Yaskawa INFORM job: DEMO_ROOF_SIDE_0625_3PAINT_54.JBI

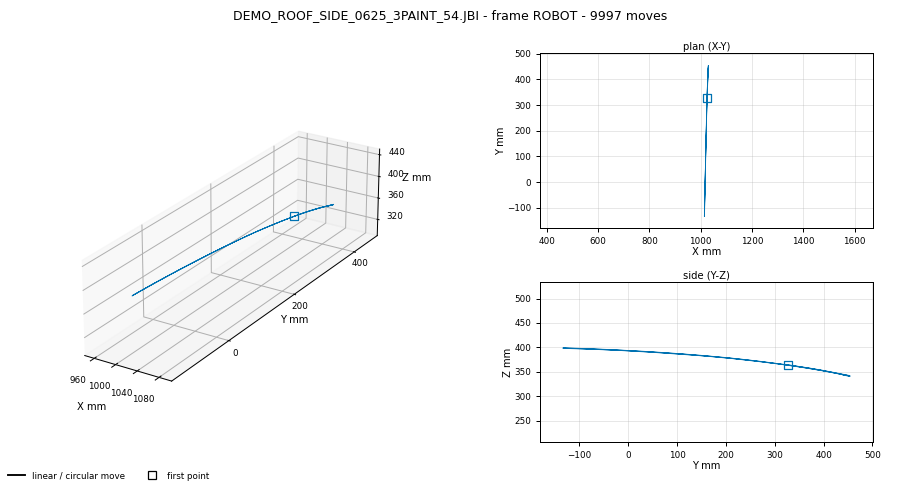
[picture p0: tool path of DEMO_ROOF_SIDE_0625_3PAINT_54.JBI in frame ROBOT, 9997 of 9997 moves have a stored position in this frame; points joined in program order, loops and branches not executed]
/JOB
//NAME DEMO_ROOF_SIDE_0625_3PAINT54
//POS
///NPOS 9997,0,0,0,0,0
///TOOL 0
///USER 0
///POSTYPE ROBOT
///RECTAN
///RCONF 1,0,0,0,0,0,0,0,0,0,0,0,0,0,0,0,0,0,0,0,0,0,0,0
C00000=1025.330,327.745,364.272,171.208,47.893,159.349
C00001=1025.337,327.993,364.236,171.213,47.892,159.350
C00002=1025.345,328.240,364.202,171.218,47.891,159.350
C00003=1025.352,328.488,364.166,171.225,47.891,159.351
C00004=1025.359,328.735,364.131,171.230,47.890,159.352
C00005=1025.365,328.982,364.095,171.237,47.889,159.352
C00006=1025.373,329.230,364.060,171.242,47.888,159.353
C00007=1025.380,329.477,364.025,171.248,47.888,159.354
C00008=1025.388,329.725,363.990,171.254,47.886,159.354
C00009=1025.395,329.972,363.954,171.260,47.886,159.355
C00010=1025.402,330.219,363.919,171.265,47.885,159.355
C00011=1025.409,330.467,363.883,171.272,47.885,159.356
C00012=1025.417,330.714,363.848,171.277,47.884,159.357
C00013=1025.424,330.961,363.813,171.284,47.883,159.358
C00014=1025.431,331.209,363.778,171.289,47.883,159.358
C00015=1025.438,331.456,363.742,171.295,47.882,159.359
C00016=1025.445,331.704,363.706,171.301,47.881,159.359
C00017=1025.453,331.951,363.672,171.307,47.880,159.360
C00018=1025.461,332.199,363.635,171.313,47.880,159.361
C00019=1025.467,332.446,363.600,171.319,47.880,159.361
C00020=1025.475,332.693,363.564,171.325,47.878,159.362
C00021=1025.482,332.941,363.529,171.331,47.878,159.363
C00022=1025.489,333.188,363.493,171.337,47.877,159.363
C00023=1025.497,333.435,363.458,171.343,47.877,159.364
C00024=1025.505,333.683,363.422,171.348,47.876,159.365
C00025=1025.512,333.929,363.386,171.355,47.876,159.365
C00026=1025.519,334.177,363.351,171.361,47.875,159.366
C00027=1025.526,334.424,363.315,171.368,47.875,159.367
C00028=1025.534,334.672,363.279,171.373,47.874,159.368
C00029=1025.540,334.920,363.242,171.380,47.873,159.368
C00030=1025.547,335.167,363.207,171.385,47.873,159.369
C00031=1025.555,335.414,363.170,171.392,47.873,159.370
C00032=1025.562,335.661,363.135,171.398,47.872,159.371
C00033=1025.574,336.048,363.078,171.407,47.871,159.372
C00034=1025.586,336.435,363.022,171.416,47.871,159.373
C00035=1025.597,336.822,362.966,171.426,47.870,159.374
C00036=1025.608,337.209,362.909,171.435,47.869,159.375
C00037=1025.616,337.456,362.873,171.442,47.869,159.376
C00038=1025.623,337.704,362.837,171.448,47.869,159.376
C00039=1025.631,337.951,362.801,171.455,47.868,159.377
C00040=1025.638,338.198,362.765,171.460,47.868,159.378
C00041=1025.646,338.446,362.728,171.467,47.867,159.379
C00042=1025.654,338.693,362.692,171.474,47.867,159.380
C00043=1025.661,338.940,362.656,171.479,47.866,159.380
C00044=1025.668,339.187,362.620,171.486,47.866,159.381
C00045=1025.676,339.435,362.584,171.492,47.866,159.382
C00046=1025.684,339.682,362.548,171.498,47.865,159.383
C00047=1025.691,339.930,362.511,171.504,47.865,159.383
C00048=1025.698,340.176,362.474,171.511,47.865,159.384
C00049=1025.706,340.423,362.438,171.517,47.865,159.385
C00050=1025.713,340.671,362.402,171.523,47.864,159.386
C00051=1025.721,340.918,362.364,171.530,47.864,159.387
C00052=1025.728,341.165,362.328,171.536,47.864,159.387
C00053=1025.735,341.412,362.292,171.543,47.864,159.388
C00054=1025.743,341.659,362.255,171.548,47.863,159.389
C00055=1025.750,341.907,362.218,171.555,47.863,159.390
C00056=1025.758,342.154,362.182,171.561,47.863,159.391
C00057=1025.765,342.401,362.145,171.568,47.863,159.392
C00058=1025.773,342.649,362.109,171.575,47.862,159.392
C00059=1025.781,342.896,362.072,171.581,47.863,159.393
C00060=1025.788,343.143,362.035,171.587,47.862,159.394
C00061=1025.796,343.390,361.998,171.593,47.862,159.395
C00062=1025.803,343.638,361.962,171.600,47.862,159.396
C00063=1025.811,343.885,361.924,171.607,47.861,159.397
C00064=1025.818,344.131,361.888,171.613,47.862,159.397
C00065=1025.825,344.379,361.851,171.619,47.861,159.398
C00066=1025.833,344.625,361.814,171.626,47.861,159.399
C00067=1025.841,344.872,361.777,171.632,47.861,159.400
C00068=1025.848,345.120,361.740,171.639,47.861,159.401
C00069=1025.856,345.367,361.703,171.645,47.861,159.402
C00070=1025.864,345.615,361.665,171.652,47.861,159.403
C00071=1025.871,345.862,361.629,171.658,47.860,159.403
C00072=1025.879,346.109,361.591,171.664,47.861,159.404
C00073=1025.887,346.356,361.555,171.671,47.861,159.405
C00074=1025.895,346.603,361.518,171.678,47.860,159.406
C00075=1025.902,346.850,361.480,171.685,47.860,159.407
C00076=1025.910,347.097,361.443,171.691,47.861,159.408
C00077=1025.917,347.345,361.406,171.698,47.860,159.409
C00078=1025.925,347.591,361.369,171.705,47.860,159.410
C00079=1025.932,347.839,361.332,171.711,47.861,159.411
C00080=1025.941,348.086,361.295,171.718,47.861,159.412
C00081=1025.948,348.333,361.257,171.725,47.860,159.412
C00082=1025.956,348.580,361.220,171.732,47.860,159.413
C00083=1025.963,348.827,361.182,171.738,47.861,159.414
C00084=1025.971,349.074,361.144,171.745,47.861,159.415
C00085=1025.979,349.321,361.107,171.752,47.861,159.416
C00086=1025.986,349.568,361.070,171.758,47.861,159.417
C00087=1025.994,349.816,361.032,171.765,47.861,159.418
C00088=1026.005,350.185,360.975,171.775,47.861,159.420
C00089=1026.016,350.531,360.923,171.784,47.861,159.421
C00090=1026.023,350.754,360.890,171.790,47.862,159.422
C00091=1026.030,350.977,360.855,171.796,47.862,159.423
C00092=1026.037,351.199,360.821,171.802,47.862,159.424
C00093=1026.044,351.423,360.787,171.809,47.862,159.424
C00094=1026.051,351.645,360.753,171.815,47.862,159.425
C00095=1026.058,351.868,360.719,171.821,47.863,159.426
C00096=1026.065,352.090,360.685,171.827,47.863,159.427
C00097=1026.074,352.338,360.648,171.834,47.863,159.428
C00098=1026.081,352.584,360.609,171.841,47.863,159.429
C00099=1026.088,352.831,360.572,171.848,47.863,159.430
C00100=1026.096,353.079,360.533,171.855,47.863,159.431
C00101=1026.104,353.325,360.496,171.861,47.864,159.432
C00102=1026.113,353.573,360.458,171.869,47.864,159.433
C00103=1026.120,353.820,360.420,171.876,47.864,159.434
C00104=1026.128,354.066,360.382,171.883,47.864,159.435
C00105=1026.136,354.314,360.345,171.890,47.865,159.436
C00106=1026.144,354.560,360.306,171.897,47.865,159.437
C00107=1026.152,354.808,360.268,171.904,47.865,159.438
C00108=1026.160,355.054,360.231,171.910,47.866,159.439
C00109=1026.168,355.302,360.192,171.917,47.866,159.440
C00110=1026.175,355.548,360.154,171.924,47.866,159.441
C00111=1026.184,355.795,360.115,171.932,47.867,159.442
C00112=1026.191,356.042,360.077,171.939,47.867,159.443
C00113=1026.199,356.289,360.038,171.946,47.868,159.445
C00114=1026.206,356.536,360.001,171.953,47.868,159.446
C00115=1026.215,356.783,359.962,171.960,47.868,159.447
C00116=1026.222,357.030,359.924,171.967,47.868,159.448
C00117=1026.230,357.277,359.885,171.975,47.869,159.449
C00118=1026.239,357.524,359.847,171.981,47.870,159.450
C00119=1026.247,357.771,359.809,171.988,47.870,159.451
C00120=1026.255,358.018,359.771,171.995,47.871,159.452
C00121=1026.263,358.265,359.732,172.002,47.871,159.453
C00122=1026.271,358.511,359.693,172.010,47.872,159.454
C00123=1026.279,358.758,359.654,172.017,47.872,159.456
C00124=1026.287,359.005,359.616,172.024,47.873,159.457
C00125=1026.295,359.252,359.578,172.031,47.873,159.458
C00126=1026.303,359.499,359.539,172.039,47.874,159.459
C00127=1026.311,359.746,359.500,172.046,47.874,159.460
C00128=1026.319,359.992,359.461,172.053,47.875,159.461
C00129=1026.327,360.239,359.423,172.060,47.875,159.462
C00130=1026.335,360.487,359.384,172.068,47.876,159.463
C00131=1026.344,360.733,359.345,172.075,47.876,159.465
C00132=1026.351,360.980,359.307,172.083,47.877,159.466
C00133=1026.359,361.227,359.267,172.090,47.878,159.467
C00134=1026.367,361.474,359.228,172.097,47.878,159.468
C00135=1026.376,361.720,359.189,172.105,47.879,159.469
C00136=1026.383,361.967,359.151,172.112,47.880,159.470
C00137=1026.391,362.214,359.111,172.119,47.880,159.472
C00138=1026.399,362.461,359.072,172.127,47.881,159.473
C00139=1026.407,362.708,359.033,172.134,47.882,159.474
C00140=1026.416,362.954,358.993,172.143,47.882,159.475
C00141=1026.423,363.202,358.954,172.150,47.883,159.476
C00142=1026.432,363.448,358.915,172.157,47.884,159.478
C00143=1026.440,363.694,358.876,172.165,47.884,159.479
C00144=1026.448,363.941,358.837,172.172,47.885,159.480
C00145=1026.456,364.188,358.798,172.180,47.886,159.481
C00146=1026.464,364.435,358.758,172.187,47.887,159.483
C00147=1026.472,364.682,358.719,172.194,47.888,159.484
C00148=1026.481,364.928,358.679,172.202,47.888,159.485
C00149=1026.489,365.155,358.644,172.209,47.889,159.486
C00150=1026.495,365.381,358.607,172.216,47.890,159.487
C00151=1026.503,365.606,358.571,172.223,47.891,159.488
C00152=1026.511,365.833,358.535,172.230,47.891,159.490
C00153=1026.518,366.059,358.499,172.237,47.892,159.491
C00154=1026.526,366.284,358.462,172.244,47.893,159.492
C00155=1026.534,366.511,358.427,172.251,47.893,159.493
C00156=1026.542,366.737,358.391,172.259,47.895,159.494
C00157=1026.549,366.984,358.351,172.266,47.895,159.496
C00158=1026.558,367.230,358.311,172.274,47.897,159.497
C00159=1026.567,367.477,358.271,172.281,47.897,159.498
C00160=1026.575,367.723,358.232,172.290,47.898,159.499
C00161=1026.583,367.970,358.192,172.297,47.899,159.501
C00162=1026.592,368.218,358.152,172.305,47.900,159.502
C00163=1026.600,368.464,358.113,172.312,47.901,159.503
C00164=1026.609,368.710,358.073,172.321,47.902,159.505
C00165=1026.617,368.957,358.033,172.328,47.903,159.506
C00166=1026.625,369.204,357.994,172.336,47.903,159.507
C00167=1026.633,369.450,357.953,172.344,47.905,159.509
C00168=1026.642,369.698,357.913,172.352,47.906,159.510
C00169=1026.650,369.943,357.873,172.360,47.907,159.511
C00170=1026.658,370.190,357.833,172.368,47.908,159.513
C00171=1026.667,370.436,357.793,172.375,47.909,159.514
C00172=1026.675,370.684,357.753,172.384,47.910,159.516
C00173=1026.683,370.930,357.712,172.392,47.911,159.517
C00174=1026.692,371.176,357.672,172.399,47.912,159.518
C00175=1026.700,371.423,357.632,172.408,47.913,159.520
C00176=1026.709,371.670,357.592,172.415,47.914,159.521
C00177=1026.717,371.916,357.551,172.423,47.915,159.522
C00178=1026.726,372.163,357.512,172.432,47.917,159.524
C00179=1026.734,372.410,357.471,172.440,47.918,159.525
C00180=1026.742,372.656,357.430,172.447,47.919,159.527
C00181=1026.752,372.903,357.390,172.456,47.920,159.528
C00182=1026.760,373.149,357.349,172.464,47.922,159.529
C00183=1026.768,373.395,357.309,172.472,47.923,159.531
C00184=1026.777,373.643,357.269,172.480,47.924,159.532
C00185=1026.785,373.889,357.228,172.488,47.926,159.534
C00186=1026.794,374.135,357.188,172.497,47.926,159.535
C00187=1026.802,374.382,357.147,172.504,47.928,159.537
C00188=1026.811,374.628,357.107,172.513,47.929,159.538
C00189=1026.820,374.875,357.066,172.521,47.930,159.540
C00190=1026.828,375.122,357.025,172.530,47.931,159.541
C00191=1026.838,375.368,356.984,172.537,47.933,159.542
C00192=1026.846,375.614,356.943,172.546,47.934,159.544
C00193=1026.855,375.861,356.903,172.554,47.935,159.545
C00194=1026.863,376.107,356.862,172.563,47.937,159.547
C00195=1026.872,376.354,356.821,172.571,47.938,159.548
C00196=1026.881,376.601,356.781,172.580,47.939,159.550
C00197=1026.890,376.846,356.739,172.588,47.941,159.551
C00198=1026.899,377.093,356.699,172.597,47.942,159.553
C00199=1026.908,377.340,356.658,172.604,47.943,159.554
C00200=1026.916,377.586,356.617,172.613,47.945,159.556
C00201=1026.925,377.833,356.576,172.622,47.946,159.558
C00202=1026.933,378.079,356.534,172.630,47.948,159.559
C00203=1026.942,378.325,356.493,172.639,47.949,159.561
C00204=1026.950,378.572,356.452,172.647,47.951,159.562
C00205=1026.959,378.818,356.410,172.656,47.952,159.564
C00206=1026.967,379.064,356.369,172.664,47.954,159.565
C00207=1026.976,379.311,356.328,172.673,47.955,159.567
C00208=1026.985,379.557,356.286,172.682,47.957,159.569
C00209=1026.994,379.794,356.247,172.690,47.958,159.570
C00210=1027.002,380.030,356.207,172.698,47.960,159.572
C00211=1027.011,380.266,356.167,172.706,47.961,159.573
C00212=1027.018,380.504,356.127,172.714,47.963,159.575
C00213=1027.028,380.741,356.086,172.723,47.964,159.576
C00214=1027.036,380.978,356.047,172.731,47.966,159.578
C00215=1027.045,381.214,356.007,172.739,47.968,159.579
C00216=1027.053,381.450,355.967,172.748,47.969,159.581
C00217=1027.062,381.696,355.925,172.757,47.970,159.583
C00218=1027.071,381.943,355.884,172.766,47.973,159.584
C00219=1027.080,382.189,355.842,172.775,47.974,159.586
C00220=1027.089,382.436,355.800,172.784,47.976,159.588
C00221=1027.098,382.682,355.759,172.793,47.977,159.589
C00222=1027.107,382.928,355.717,172.801,47.979,159.591
C00223=1027.116,383.175,355.675,172.810,47.981,159.593
C00224=1027.125,383.421,355.633,172.819,47.982,159.594
C00225=1027.134,383.667,355.591,172.828,47.984,159.596
C00226=1027.143,383.913,355.549,172.837,47.986,159.598
C00227=1027.152,384.159,355.508,172.845,47.988,159.599
C00228=1027.161,384.407,355.465,172.854,47.989,159.601
C00229=1027.171,384.652,355.423,172.864,47.991,159.603
C00230=1027.180,384.899,355.381,172.873,47.993,159.604
C00231=1027.188,385.145,355.340,172.882,47.995,159.606
C00232=1027.198,385.391,355.297,172.891,47.996,159.608
C00233=1027.207,385.637,355.255,172.900,47.998,159.610
C00234=1027.216,385.884,355.213,172.909,48.001,159.611
C00235=1027.226,386.130,355.172,172.918,48.002,159.613
C00236=1027.235,386.375,355.129,172.927,48.004,159.615
C00237=1027.244,386.622,355.087,172.936,48.006,159.617
C00238=1027.253,386.869,355.044,172.946,48.008,159.618
C00239=1027.263,387.114,355.002,172.955,48.010,159.620
C00240=1027.272,387.360,354.959,172.964,48.012,159.622
C00241=1027.280,387.607,354.917,172.974,48.014,159.624
C00242=1027.290,387.853,354.874,172.983,48.016,159.626
C00243=1027.299,388.099,354.832,172.992,48.018,159.628
C00244=1027.308,388.345,354.789,173.001,48.019,159.629
C00245=1027.318,388.591,354.746,173.011,48.021,159.631
C00246=1027.327,388.837,354.703,173.020,48.023,159.633
C00247=1027.337,389.084,354.661,173.030,48.025,159.635
C00248=1027.346,389.329,354.618,173.039,48.027,159.637
C00249=1027.355,389.575,354.576,173.049,48.030,159.639
C00250=1027.364,389.822,354.532,173.058,48.032,159.640
C00251=1027.373,390.068,354.490,173.067,48.034,159.642
C00252=1027.383,390.314,354.446,173.077,48.036,159.644
C00253=1027.392,390.559,354.403,173.086,48.038,159.646
C00254=1027.402,390.806,354.360,173.097,48.040,159.648
C00255=1027.410,391.052,354.317,173.106,48.042,159.650
C00256=1027.421,391.298,354.274,173.115,48.045,159.652
C00257=1027.430,391.543,354.232,173.125,48.047,159.654
C00258=1027.439,391.790,354.188,173.135,48.049,159.656
C00259=1027.448,392.035,354.145,173.144,48.051,159.658
C00260=1027.458,392.282,354.102,173.155,48.053,159.660
C00261=1027.468,392.528,354.058,173.164,48.055,159.661
C00262=1027.477,392.774,354.016,173.174,48.058,159.664
C00263=1027.486,393.020,353.972,173.183,48.061,159.666
C00264=1027.496,393.266,353.928,173.193,48.063,159.667
C00265=1027.506,393.512,353.885,173.203,48.065,159.669
C00266=1027.515,393.758,353.841,173.213,48.067,159.671
C00267=1027.525,394.004,353.797,173.222,48.070,159.673
C00268=1027.534,394.250,353.755,173.232,48.072,159.675
C00269=1027.544,394.513,353.707,173.243,48.074,159.678
C00270=1027.555,394.776,353.661,173.254,48.077,159.680
C00271=1027.565,395.040,353.615,173.265,48.079,159.682
C00272=1027.575,395.303,353.567,173.275,48.082,159.684
C00273=1027.585,395.549,353.523,173.285,48.084,159.686
C00274=1027.594,395.795,353.480,173.295,48.087,159.688
C00275=1027.604,396.041,353.435,173.305,48.089,159.690
C00276=1027.614,396.287,353.392,173.315,48.092,159.692
C00277=1027.623,396.533,353.348,173.326,48.094,159.694
C00278=1027.633,396.779,353.304,173.336,48.097,159.697
C00279=1027.643,397.025,353.260,173.346,48.100,159.699
C00280=1027.653,397.270,353.216,173.356,48.102,159.701
C00281=1027.663,397.516,353.172,173.366,48.105,159.703
C00282=1027.673,397.762,353.128,173.377,48.107,159.705
C00283=1027.683,398.007,353.084,173.387,48.109,159.707
C00284=1027.692,398.253,353.039,173.398,48.112,159.709
C00285=1027.702,398.499,352.996,173.407,48.115,159.711
C00286=1027.712,398.745,352.951,173.418,48.117,159.713
C00287=1027.721,398.991,352.907,173.428,48.120,159.716
C00288=1027.732,399.236,352.863,173.439,48.122,159.718
C00289=1027.741,399.482,352.818,173.449,48.125,159.720
C00290=1027.751,399.728,352.773,173.460,48.128,159.722
C00291=1027.761,399.974,352.729,173.471,48.130,159.725
C00292=1027.772,400.219,352.684,173.481,48.134,159.727
C00293=1027.781,400.465,352.640,173.491,48.136,159.729
C00294=1027.791,400.711,352.595,173.501,48.139,159.731
C00295=1027.801,400.957,352.550,173.513,48.142,159.733
C00296=1027.811,401.203,352.505,173.523,48.144,159.736
C00297=1027.820,401.448,352.461,173.533,48.147,159.738
C00298=1027.831,401.693,352.416,173.544,48.150,159.740
C00299=1027.841,401.939,352.371,173.555,48.153,159.742
C00300=1027.851,402.185,352.326,173.566,48.155,159.745
C00301=1027.861,402.431,352.282,173.577,48.159,159.747
C00302=1027.871,402.677,352.236,173.588,48.161,159.749
C00303=1027.881,402.922,352.192,173.599,48.164,159.752
C00304=1027.891,403.168,352.146,173.609,48.167,159.754
C00305=1027.901,403.413,352.101,173.620,48.170,159.756
C00306=1027.911,403.659,352.056,173.631,48.173,159.759
C00307=1027.921,403.905,352.011,173.642,48.176,159.761
C00308=1027.931,404.150,351.965,173.653,48.179,159.763
C00309=1027.941,404.396,351.920,173.664,48.182,159.766
C00310=1027.951,404.641,351.875,173.674,48.185,159.768
C00311=1027.962,404.887,351.829,173.686,48.188,159.771
C00312=1027.972,405.133,351.783,173.697,48.191,159.773
C00313=1027.982,405.378,351.739,173.708,48.194,159.775
C00314=1027.993,405.624,351.693,173.719,48.197,159.778
C00315=1028.003,405.870,351.648,173.730,48.200,159.780
C00316=1028.013,406.115,351.602,173.742,48.203,159.783
C00317=1028.024,406.361,351.556,173.753,48.206,159.785
C00318=1028.034,406.606,351.510,173.764,48.209,159.787
C00319=1028.044,406.852,351.465,173.776,48.212,159.790
C00320=1028.055,407.097,351.419,173.787,48.216,159.793
C00321=1028.065,407.343,351.374,173.798,48.219,159.795
C00322=1028.076,407.589,351.328,173.810,48.222,159.797
C00323=1028.086,407.834,351.282,173.821,48.225,159.800
C00324=1028.097,408.080,351.236,173.833,48.228,159.802
C00325=1028.107,408.325,351.190,173.844,48.232,159.805
C00326=1028.118,408.570,351.144,173.855,48.235,159.807
C00327=1028.128,408.816,351.098,173.867,48.237,159.810
C00328=1028.139,409.061,351.053,173.879,48.241,159.812
C00329=1028.151,409.347,350.999,173.892,48.245,159.815
C00330=1028.164,409.633,350.945,173.906,48.249,159.818
C00331=1028.176,409.918,350.891,173.919,48.253,159.821
C00332=1028.189,410.203,350.838,173.933,48.256,159.824
C00333=1028.199,410.448,350.791,173.945,48.260,159.827
C00334=1028.210,410.693,350.745,173.956,48.263,159.830
C00335=1028.221,410.939,350.699,173.969,48.267,159.832
C00336=1028.231,411.184,350.652,173.980,48.270,159.835
C00337=1028.241,411.430,350.606,173.992,48.273,159.838
C00338=1028.252,411.675,350.559,174.005,48.277,159.840
C00339=1028.263,411.921,350.511,174.016,48.281,159.843
C00340=1028.274,412.166,350.466,174.028,48.284,159.846
C00341=1028.284,412.412,350.418,174.041,48.288,159.848
C00342=1028.295,412.657,350.372,174.052,48.291,159.851
C00343=1028.306,412.902,350.325,174.065,48.294,159.854
C00344=1028.317,413.148,350.278,174.077,48.298,159.856
C00345=1028.327,413.393,350.231,174.089,48.302,159.859
C00346=1028.339,413.638,350.184,174.101,48.305,159.862
C00347=1028.349,413.884,350.137,174.114,48.308,159.865
C00348=1028.360,414.129,350.090,174.125,48.312,159.867
C00349=1028.372,414.374,350.043,174.138,48.316,159.870
C00350=1028.382,414.620,349.996,174.150,48.319,159.873
C00351=1028.393,414.865,349.949,174.163,48.324,159.876
C00352=1028.405,415.110,349.902,174.175,48.327,159.879
C00353=1028.415,415.356,349.854,174.188,48.331,159.882
C00354=1028.426,415.601,349.807,174.200,48.334,159.884
C00355=1028.438,415.846,349.760,174.212,48.338,159.887
C00356=1028.449,416.092,349.712,174.225,48.342,159.890
C00357=1028.460,416.337,349.665,174.238,48.346,159.893
C00358=1028.471,416.582,349.617,174.251,48.349,159.896
C00359=1028.482,416.826,349.570,174.263,48.353,159.899
C00360=1028.493,417.072,349.522,174.276,48.357,159.902
C00361=1028.504,417.318,349.474,174.289,48.361,159.905
C00362=1028.516,417.563,349.426,174.302,48.365,159.908
C00363=1028.526,417.807,349.378,174.314,48.369,159.910
C00364=1028.538,418.053,349.331,174.327,48.373,159.913
C00365=1028.549,418.298,349.283,174.340,48.377,159.916
C00366=1028.560,418.544,349.235,174.353,48.381,159.919
C00367=1028.571,418.788,349.187,174.366,48.384,159.922
C00368=1028.583,419.033,349.139,174.379,48.388,159.925
C00369=1028.594,419.279,349.091,174.392,48.392,159.928
C00370=1028.605,419.524,349.043,174.406,48.396,159.931
C00371=1028.617,419.769,348.994,174.419,48.400,159.934
C00372=1028.629,420.014,348.946,174.432,48.405,159.938
C00373=1028.640,420.259,348.898,174.445,48.409,159.941
C00374=1028.651,420.504,348.850,174.459,48.413,159.944
C00375=1028.663,420.749,348.801,174.472,48.417,159.947
C00376=1028.674,420.994,348.753,174.485,48.420,159.950
C00377=1028.686,421.239,348.705,174.498,48.425,159.953
C00378=1028.697,421.484,348.656,174.512,48.429,159.956
C00379=1028.709,421.729,348.607,174.526,48.433,159.959
C00380=1028.721,421.974,348.559,174.539,48.437,159.962
C00381=1028.733,422.219,348.510,174.553,48.442,159.966
C00382=1028.744,422.465,348.462,174.566,48.446,159.969
C00383=1028.755,422.709,348.413,174.580,48.450,159.972
C00384=1028.768,422.954,348.364,174.594,48.454,159.975
C00385=1028.779,423.199,348.315,174.607,48.459,159.978
C00386=1028.791,423.444,348.266,174.622,48.462,159.982
C00387=1028.802,423.689,348.217,174.635,48.467,159.985
C00388=1028.814,423.934,348.168,174.649,48.471,159.988
C00389=1028.828,424.230,348.109,174.666,48.476,159.992
C00390=1028.842,424.525,348.050,174.683,48.482,159.996
C00391=1028.857,424.821,347.990,174.699,48.488,160.000
C00392=1028.871,425.117,347.931,174.717,48.493,160.004
C00393=1028.883,425.361,347.881,174.730,48.497,160.007
C00394=1028.895,425.606,347.832,174.745,48.501,160.011
C00395=1028.907,425.851,347.783,174.759,48.505,160.014
C00396=1028.919,426.096,347.733,174.773,48.510,160.018
C00397=1028.932,426.341,347.684,174.788,48.515,160.021
C00398=1028.943,426.585,347.634,174.802,48.520,160.024
C00399=1028.956,426.830,347.584,174.817,48.524,160.028
C00400=1028.967,427.076,347.534,174.831,48.528,160.031
C00401=1028.979,427.320,347.484,174.846,48.533,160.035
C00402=1028.991,427.565,347.434,174.860,48.538,160.038
C00403=1029.003,427.810,347.384,174.875,48.543,160.042
C00404=1029.015,428.054,347.334,174.890,48.547,160.045
C00405=1029.027,428.298,347.284,174.905,48.552,160.049
C00406=1029.040,428.543,347.234,174.919,48.556,160.052
C00407=1029.052,428.788,347.184,174.933,48.561,160.056
C00408=1029.064,429.033,347.134,174.948,48.566,160.059
C00409=1029.076,429.278,347.084,174.963,48.571,160.063
C00410=1029.089,429.522,347.033,174.978,48.575,160.066
C00411=1029.101,429.766,346.983,174.993,48.580,160.070
C00412=1029.113,430.011,346.933,175.008,48.585,160.074
C00413=1029.125,430.255,346.882,175.023,48.590,160.077
C00414=1029.137,430.500,346.832,175.038,48.595,160.081
C00415=1029.151,430.745,346.781,175.053,48.599,160.085
C00416=1029.163,430.990,346.730,175.070,48.604,160.088
C00417=1029.175,431.234,346.680,175.085,48.609,160.092
C00418=1029.188,431.479,346.630,175.100,48.614,160.096
C00419=1029.200,431.723,346.579,175.115,48.619,160.099
C00420=1029.213,431.967,346.528,175.130,48.624,160.103
C00421=1029.226,432.212,346.477,175.146,48.629,160.107
C00422=1029.239,432.457,346.426,175.162,48.634,160.111
C00423=1029.251,432.701,346.376,175.177,48.639,160.114
C00424=1029.264,432.946,346.325,175.193,48.644,160.118
C00425=1029.277,433.190,346.274,175.209,48.649,160.122
C00426=1029.289,433.435,346.222,175.225,48.654,160.126
C00427=1029.302,433.679,346.171,175.240,48.659,160.130
C00428=1029.315,433.923,346.120,175.257,48.664,160.134
C00429=1029.328,434.168,346.069,175.272,48.669,160.137
C00430=1029.340,434.412,346.016,175.289,48.674,160.141
C00431=1029.354,434.657,345.965,175.304,48.679,160.145
C00432=1029.367,434.901,345.914,175.321,48.685,160.149
C00433=1029.380,435.146,345.863,175.336,48.690,160.153
C00434=1029.392,435.389,345.810,175.352,48.695,160.157
C00435=1029.405,435.634,345.759,175.369,48.700,160.161
C00436=1029.419,435.879,345.707,175.385,48.706,160.165
C00437=1029.431,436.123,345.655,175.401,48.711,160.169
C00438=1029.444,436.367,345.603,175.418,48.716,160.173
C00439=1029.458,436.611,345.551,175.435,48.721,160.177
C00440=1029.471,436.856,345.499,175.451,48.727,160.181
C00441=1029.484,437.099,345.447,175.468,48.732,160.185
C00442=1029.497,437.344,345.395,175.484,48.738,160.190
C00443=1029.510,437.588,345.343,175.501,48.743,160.194
C00444=1029.524,437.832,345.291,175.517,48.748,160.198
C00445=1029.536,438.077,345.239,175.534,48.754,160.202
C00446=1029.550,438.321,345.186,175.552,48.759,160.206
C00447=1029.564,438.565,345.134,175.569,48.765,160.210
C00448=1029.576,438.810,345.082,175.586,48.770,160.215
C00449=1029.590,439.053,345.029,175.603,48.776,160.219
C00450=1029.604,439.296,344.977,175.620,48.781,160.223
C00451=1029.617,439.539,344.925,175.637,48.787,160.227
C00452=1029.630,439.783,344.871,175.654,48.792,160.231
C00453=1029.643,440.026,344.819,175.672,48.798,160.236
C00454=1029.657,440.270,344.767,175.689,48.803,160.240
C00455=1029.671,440.512,344.714,175.706,48.809,160.244
C00456=1029.684,440.756,344.661,175.724,48.815,160.249
C00457=1029.697,441.000,344.608,175.741,48.821,160.253
C00458=1029.712,441.244,344.555,175.759,48.826,160.257
C00459=1029.725,441.488,344.502,175.777,48.832,160.262
C00460=1029.739,441.732,344.449,175.795,48.837,160.266
C00461=1029.753,441.976,344.395,175.812,48.844,160.271
C00462=1029.767,442.219,344.342,175.831,48.849,160.275
C00463=1029.780,442.464,344.289,175.848,48.856,160.280
C00464=1029.794,442.707,344.235,175.866,48.861,160.284
C00465=1029.809,442.950,344.182,175.884,48.867,160.289
C00466=1029.823,443.193,344.129,175.903,48.872,160.293
C00467=1029.837,443.436,344.077,175.920,48.878,160.298
C00468=1029.852,443.681,344.024,175.939,48.884,160.302
C00469=1029.867,443.923,343.971,175.957,48.890,160.307
C00470=1029.884,444.167,343.920,175.976,48.895,160.311
C00471=1029.900,444.410,343.868,175.994,48.901,160.316
C00472=1029.918,444.655,343.818,176.013,48.906,160.320
C00473=1029.935,444.898,343.768,176.032,48.911,160.325
C00474=1029.952,445.142,343.718,176.050,48.917,160.329
C00475=1029.971,445.386,343.668,176.069,48.922,160.334
C00476=1029.990,445.630,343.619,176.088,48.926,160.338
C00477=1030.009,445.873,343.570,176.108,48.932,160.343
C00478=1030.029,446.118,343.522,176.127,48.936,160.347
C00479=1030.049,446.362,343.474,176.146,48.941,160.351
C00480=1030.070,446.607,343.427,176.165,48.946,160.356
C00481=1030.093,446.877,343.374,176.186,48.951,160.361
C00482=1030.118,447.148,343.322,176.208,48.956,160.366
C00483=1030.143,447.418,343.271,176.230,48.961,160.371
C00484=1030.169,447.689,343.220,176.251,48.966,160.375
C00485=1030.191,447.933,343.175,176.271,48.971,160.380
C00486=1030.216,448.178,343.131,176.291,48.975,160.384
C00487=1030.240,448.423,343.086,176.311,48.979,160.389
C00488=1030.265,448.668,343.042,176.331,48.984,160.393
C00489=1030.290,448.913,342.998,176.351,48.988,160.397
C00490=1030.316,449.158,342.955,176.372,48.992,160.402
C00491=1030.342,449.403,342.913,176.392,48.995,160.406
C00492=1030.369,449.648,342.870,176.413,48.999,160.411
C00493=1030.397,449.893,342.828,176.433,49.004,160.415
C00494=1030.424,450.139,342.786,176.453,49.007,160.419
C00495=1030.453,450.384,342.744,176.474,49.011,160.424
C00496=1030.481,450.629,342.703,176.495,49.015,160.428
C00497=1030.511,450.875,342.663,176.515,49.018,160.432
C00498=1030.540,451.120,342.624,176.536,49.022,160.437
C00499=1030.570,451.366,342.584,176.557,49.025,160.441
C00500=1030.601,451.611,342.544,176.579,49.029,160.445
C00501=1030.633,451.857,342.506,176.599,49.032,160.450
C00502=1030.665,452.103,342.467,176.621,49.035,160.454
C00503=1030.696,452.348,342.429,176.643,49.038,160.458
C00504=1030.729,452.593,342.392,176.664,49.042,160.463
C00505=1030.763,452.839,342.355,176.685,49.045,160.467
C00506=1030.796,453.086,342.318,176.706,49.048,160.471
C00507=1030.831,453.331,342.281,176.728,49.051,160.476
C00508=1030.885,453.721,342.225,176.763,49.055,160.482
C00509=1030.606,453.791,341.892,176.767,49.118,160.503
C00510=1030.556,453.443,341.942,176.736,49.114,160.497
C00511=1030.523,453.198,341.978,176.713,49.112,160.492
C00512=1030.488,452.952,342.015,176.692,49.109,160.488
C00513=1030.455,452.706,342.052,176.670,49.106,160.484
C00514=1030.422,452.461,342.089,176.648,49.103,160.479
C00515=1030.389,452.215,342.127,176.627,49.100,160.475
C00516=1030.357,451.970,342.165,176.606,49.096,160.471
C00517=1030.326,451.724,342.203,176.584,49.093,160.467
C00518=1030.295,451.478,342.242,176.564,49.090,160.462
C00519=1030.264,451.233,342.282,176.542,49.087,160.458
C00520=1030.234,450.987,342.321,176.522,49.083,160.454
C00521=1030.205,450.742,342.361,176.501,49.080,160.449
C00522=1030.176,450.497,342.402,176.480,49.076,160.445
C00523=1030.148,450.251,342.443,176.459,49.072,160.440
C00524=1030.119,450.006,342.485,176.439,49.069,160.436
C00525=1030.092,449.760,342.526,176.418,49.065,160.432
C00526=1030.065,449.515,342.569,176.397,49.061,160.427
C00527=1030.038,449.270,342.612,176.377,49.058,160.423
C00528=1030.012,449.025,342.654,176.356,49.054,160.419
C00529=1029.986,448.780,342.698,176.336,49.049,160.414
C00530=1029.962,448.535,342.742,176.317,49.046,160.410
C00531=1029.936,448.290,342.786,176.296,49.042,160.406
C00532=1029.912,448.045,342.831,176.276,49.037,160.401
C00533=1029.888,447.801,342.876,176.256,49.033,160.397
C00534=1029.866,447.556,342.921,176.237,49.029,160.392
C00535=1029.842,447.311,342.967,176.217,49.024,160.388
C00536=1029.821,447.067,343.014,176.197,49.020,160.383
C00537=1029.798,446.822,343.061,176.178,49.015,160.379
C00538=1029.777,446.577,343.107,176.158,49.011,160.375
C00539=1029.756,446.333,343.155,176.139,49.006,160.370
C00540=1029.736,446.089,343.203,176.120,49.001,160.366
C00541=1029.717,445.845,343.251,176.101,48.997,160.361
C00542=1029.697,445.601,343.300,176.081,48.992,160.357
C00543=1029.678,445.357,343.349,176.062,48.986,160.352
C00544=1029.659,445.113,343.399,176.043,48.982,160.348
C00545=1029.641,444.869,343.448,176.025,48.977,160.344
C00546=1029.624,444.625,343.498,176.006,48.971,160.339
C00547=1029.607,444.382,343.550,175.988,48.966,160.335
C00548=1029.590,444.138,343.601,175.968,48.961,160.330
C00549=1029.575,443.894,343.653,175.950,48.956,160.326
C00550=1029.559,443.651,343.704,175.932,48.950,160.321
C00551=1029.544,443.407,343.756,175.913,48.944,160.317
C00552=1029.529,443.165,343.809,175.895,48.939,160.312
C00553=1029.515,442.922,343.862,175.877,48.933,160.308
C00554=1029.501,442.679,343.916,175.858,48.927,160.303
C00555=1029.487,442.434,343.969,175.841,48.921,160.299
C00556=1029.473,442.190,344.022,175.823,48.916,160.294
C00557=1029.459,441.946,344.076,175.804,48.910,160.290
C00558=1029.446,441.703,344.129,175.787,48.905,160.285
C00559=1029.432,441.458,344.182,175.769,48.899,160.281
C00560=1029.418,441.214,344.235,175.751,48.893,160.276
C00561=1029.405,440.970,344.288,175.733,48.887,160.272
C00562=1029.391,440.722,344.342,175.715,48.882,160.268
C00563=1029.377,440.473,344.396,175.697,48.876,160.263
C00564=1029.363,440.225,344.450,175.680,48.871,160.259
C00565=1029.349,439.976,344.504,175.662,48.865,160.254
C00566=1029.334,439.712,344.561,175.643,48.859,160.250
C00567=1029.320,439.448,344.618,175.625,48.853,160.245
C00568=1029.305,439.182,344.676,175.606,48.847,160.241
C00569=1029.290,438.917,344.733,175.587,48.841,160.236
C00570=1029.277,438.673,344.785,175.570,48.836,160.232
C00571=1029.264,438.429,344.838,175.553,48.831,160.228
C00572=1029.250,438.185,344.890,175.536,48.825,160.223
C00573=1029.237,437.940,344.942,175.519,48.820,160.219
C00574=1029.224,437.696,344.995,175.502,48.814,160.215
C00575=1029.210,437.452,345.047,175.486,48.809,160.211
C00576=1029.198,437.208,345.099,175.469,48.804,160.207
C00577=1029.184,436.964,345.151,175.452,48.798,160.203
C00578=1029.171,436.720,345.203,175.436,48.793,160.199
C00579=1029.158,436.475,345.255,175.419,48.788,160.195
C00580=1029.144,436.231,345.307,175.402,48.783,160.191
C00581=1029.132,435.987,345.359,175.386,48.778,160.186
C00582=1029.119,435.743,345.411,175.369,48.772,160.182
C00583=1029.106,435.498,345.462,175.353,48.767,160.178
C00584=1029.093,435.254,345.514,175.337,48.762,160.175
C00585=1029.080,435.009,345.566,175.320,48.757,160.171
C00586=1029.067,434.765,345.617,175.305,48.751,160.167
C00587=1029.054,434.520,345.668,175.288,48.747,160.163
C00588=1029.041,434.277,345.720,175.272,48.742,160.159
C00589=1029.029,434.032,345.772,175.256,48.736,160.155
C00590=1029.016,433.787,345.822,175.240,48.732,160.151
C00591=1029.002,433.543,345.874,175.225,48.727,160.147
C00592=1028.990,433.299,345.925,175.208,48.722,160.143
C00593=1028.977,433.054,345.976,175.193,48.716,160.139
C00594=1028.964,432.810,346.027,175.177,48.711,160.136
C00595=1028.952,432.565,346.079,175.162,48.707,160.132
C00596=1028.939,432.320,346.130,175.145,48.702,160.128
C00597=1028.927,432.076,346.180,175.130,48.697,160.124
C00598=1028.914,431.831,346.231,175.115,48.692,160.121
C00599=1028.901,431.587,346.281,175.098,48.687,160.117
C00600=1028.888,431.342,346.333,175.083,48.683,160.113
C00601=1028.876,431.097,346.383,175.068,48.678,160.109
C00602=1028.863,430.853,346.433,175.053,48.673,160.106
C00603=1028.851,430.608,346.484,175.038,48.668,160.102
C00604=1028.838,430.364,346.534,175.022,48.664,160.099
C00605=1028.826,430.119,346.584,175.007,48.659,160.095
C00606=1028.813,429.875,346.635,174.992,48.654,160.091
C00607=1028.801,429.630,346.685,174.977,48.649,160.088
C00608=1028.789,429.386,346.735,174.962,48.645,160.084
C00609=1028.776,429.141,346.786,174.947,48.640,160.081
C00610=1028.764,428.897,346.836,174.932,48.636,160.077
C00611=1028.751,428.652,346.886,174.917,48.631,160.073
C00612=1028.740,428.407,346.937,174.902,48.626,160.070
C00613=1028.728,428.162,346.987,174.887,48.622,160.066
C00614=1028.716,427.918,347.037,174.873,48.617,160.063
C00615=1028.704,427.673,347.087,174.859,48.612,160.059
C00616=1028.692,427.429,347.137,174.844,48.608,160.056
C00617=1028.679,427.184,347.187,174.829,48.603,160.052
C00618=1028.667,426.938,347.236,174.814,48.599,160.049
C00619=1028.656,426.694,347.286,174.801,48.594,160.046
C00620=1028.643,426.449,347.336,174.786,48.590,160.042
C00621=1028.631,426.204,347.386,174.771,48.586,160.039
C00622=1028.620,425.960,347.435,174.756,48.581,160.035
C00623=1028.608,425.714,347.485,174.743,48.577,160.032
C00624=1028.596,425.470,347.533,174.728,48.572,160.029
C00625=1028.583,425.225,347.583,174.715,48.568,160.025
C00626=1028.569,424.927,347.643,174.697,48.563,160.021
C00627=1028.554,424.630,347.703,174.680,48.558,160.017
C00628=1028.540,424.331,347.763,174.663,48.552,160.013
C00629=1028.525,424.033,347.823,174.645,48.547,160.009
C00630=1028.514,423.788,347.872,174.632,48.543,160.006
C00631=1028.503,423.544,347.921,174.618,48.539,160.003
C00632=1028.491,423.299,347.970,174.604,48.534,159.999
C00633=1028.479,423.053,348.019,174.591,48.530,159.996
C00634=1028.468,422.809,348.068,174.576,48.526,159.993
C00635=1028.456,422.564,348.116,174.563,48.522,159.990
C00636=1028.444,422.319,348.165,174.549,48.517,159.987
C00637=1028.432,422.073,348.214,174.535,48.514,159.983
C00638=1028.420,421.829,348.262,174.522,48.509,159.980
C00639=1028.409,421.584,348.311,174.508,48.505,159.977
C00640=1028.398,421.339,348.360,174.495,48.501,159.974
C00641=1028.386,421.094,348.407,174.481,48.497,159.971
C00642=1028.375,420.849,348.456,174.467,48.493,159.968
C00643=1028.362,420.603,348.505,174.454,48.489,159.965
C00644=1028.351,420.358,348.553,174.441,48.485,159.962
C00645=1028.340,420.113,348.602,174.428,48.481,159.959
C00646=1028.328,419.868,348.650,174.415,48.477,159.956
C00647=1028.317,419.623,348.698,174.402,48.474,159.953
C00648=1028.305,419.378,348.745,174.388,48.470,159.949
C00649=1028.294,419.133,348.794,174.375,48.466,159.946
C00650=1028.283,418.888,348.842,174.362,48.462,159.943
C00651=1028.271,418.643,348.890,174.349,48.458,159.940
C00652=1028.260,418.397,348.938,174.336,48.454,159.938
C00653=1028.249,418.152,348.986,174.323,48.450,159.934
C00654=1028.238,417.908,349.033,174.310,48.446,159.931
C00655=1028.227,417.662,349.082,174.297,48.443,159.929
C00656=1028.215,417.417,349.129,174.284,48.439,159.926
C00657=1028.204,417.171,349.177,174.271,48.435,159.923
C00658=1028.194,416.927,349.225,174.258,48.431,159.920
C00659=1028.182,416.681,349.273,174.246,48.428,159.917
C00660=1028.171,416.435,349.320,174.233,48.424,159.914
C00661=1028.160,416.191,349.368,174.220,48.420,159.911
C00662=1028.149,415.945,349.415,174.207,48.417,159.908
C00663=1028.138,415.701,349.463,174.195,48.412,159.905
C00664=1028.126,415.455,349.509,174.182,48.409,159.902
C00665=1028.116,415.209,349.557,174.169,48.405,159.900
C00666=1028.104,414.965,349.604,174.158,48.402,159.897
C00667=1028.093,414.719,349.651,174.145,48.398,159.894
C00668=1028.083,414.474,349.699,174.132,48.395,159.891
C00669=1028.072,414.229,349.745,174.120,48.391,159.888
C00670=1028.060,413.983,349.792,174.108,48.388,159.886
C00671=1028.050,413.738,349.839,174.095,48.384,159.883
C00672=1028.038,413.492,349.886,174.083,48.381,159.880
C00673=1028.028,413.247,349.933,174.070,48.377,159.877
C00674=1028.017,413.002,349.980,174.059,48.373,159.875
C00675=1028.006,412.756,350.027,174.046,48.370,159.872
C00676=1027.995,412.511,350.074,174.034,48.367,159.869
C00677=1027.985,412.266,350.121,174.022,48.364,159.867
C00678=1027.974,412.020,350.167,174.010,48.360,159.864
C00679=1027.963,411.775,350.214,173.999,48.357,159.861
C00680=1027.952,411.529,350.261,173.986,48.353,159.859
C00681=1027.941,411.285,350.308,173.974,48.350,159.856
C00682=1027.931,411.039,350.354,173.962,48.346,159.853
C00683=1027.921,410.794,350.401,173.950,48.343,159.851
C00684=1027.910,410.548,350.447,173.939,48.340,159.848
C00685=1027.899,410.303,350.493,173.927,48.336,159.846
C00686=1027.887,410.015,350.548,173.913,48.333,159.842
C00687=1027.874,409.728,350.602,173.899,48.329,159.839
C00688=1027.862,409.440,350.656,173.885,48.325,159.836
C00689=1027.849,409.153,350.710,173.872,48.321,159.833
C00690=1027.839,408.907,350.756,173.861,48.318,159.831
C00691=1027.828,408.661,350.801,173.848,48.315,159.828
C00692=1027.817,408.416,350.847,173.837,48.312,159.826
C00693=1027.807,408.170,350.893,173.825,48.309,159.823
C00694=1027.796,407.925,350.939,173.814,48.305,159.821
C00695=1027.785,407.679,350.985,173.803,48.303,159.818
C00696=1027.775,407.433,351.031,173.790,48.300,159.816
C00697=1027.764,407.188,351.077,173.779,48.296,159.813
C00698=1027.754,406.943,351.122,173.768,48.294,159.811
C00699=1027.744,406.697,351.168,173.756,48.290,159.808
C00700=1027.733,406.451,351.213,173.745,48.287,159.806
C00701=1027.723,406.205,351.259,173.734,48.284,159.803
C00702=1027.713,405.961,351.305,173.723,48.281,159.801
C00703=1027.702,405.714,351.350,173.711,48.278,159.799
C00704=1027.692,405.469,351.396,173.700,48.275,159.796
C00705=1027.682,405.224,351.442,173.689,48.272,159.794
C00706=1027.671,404.978,351.487,173.678,48.269,159.791
C00707=1027.661,404.733,351.532,173.667,48.267,159.789
C00708=1027.651,404.487,351.577,173.656,48.264,159.787
C00709=1027.641,404.241,351.622,173.644,48.261,159.784
C00710=1027.631,403.995,351.668,173.634,48.257,159.782
C00711=1027.621,403.750,351.713,173.623,48.255,159.780
C00712=1027.610,403.504,351.759,173.612,48.252,159.777
C00713=1027.601,403.259,351.804,173.601,48.249,159.775
C00714=1027.590,403.013,351.849,173.590,48.246,159.773
C00715=1027.581,402.767,351.894,173.579,48.244,159.770
C00716=1027.570,402.521,351.939,173.569,48.241,159.768
C00717=1027.560,402.276,351.985,173.558,48.238,159.766
C00718=1027.550,402.031,352.029,173.547,48.235,159.763
C00719=1027.541,401.785,352.074,173.535,48.232,159.761
C00720=1027.530,401.539,352.119,173.526,48.230,159.759
C00721=1027.521,401.293,352.164,173.515,48.227,159.757
C00722=1027.511,401.047,352.208,173.504,48.224,159.754
C00723=1027.500,400.801,352.253,173.493,48.222,159.752
C00724=1027.491,400.556,352.298,173.483,48.219,159.750
C00725=1027.481,400.310,352.343,173.472,48.216,159.748
C00726=1027.471,400.065,352.387,173.461,48.214,159.745
C00727=1027.462,399.819,352.431,173.451,48.211,159.743
C00728=1027.451,399.573,352.476,173.440,48.208,159.741
C00729=1027.441,399.327,352.521,173.430,48.205,159.739
C00730=1027.432,399.081,352.565,173.419,48.203,159.737
C00731=1027.421,398.836,352.609,173.409,48.201,159.735
C00732=1027.412,398.590,352.653,173.399,48.198,159.732
C00733=1027.402,398.344,352.698,173.388,48.196,159.730
C00734=1027.392,398.098,352.742,173.378,48.193,159.728
C00735=1027.382,397.852,352.786,173.367,48.191,159.726
C00736=1027.373,397.607,352.831,173.358,48.188,159.724
C00737=1027.363,397.361,352.874,173.347,48.185,159.722
C00738=1027.353,397.115,352.918,173.337,48.183,159.720
C00739=1027.343,396.869,352.962,173.326,48.181,159.717
C00740=1027.333,396.623,353.007,173.316,48.178,159.715
C00741=1027.323,396.378,353.050,173.306,48.176,159.713
C00742=1027.314,396.131,353.094,173.296,48.173,159.711
C00743=1027.304,395.885,353.138,173.285,48.171,159.709
C00744=1027.294,395.639,353.182,173.276,48.169,159.707
C00745=1027.285,395.393,353.226,173.265,48.167,159.705
C00746=1027.275,395.128,353.273,173.254,48.164,159.703
C00747=1027.264,394.863,353.320,173.244,48.161,159.701
C00748=1027.254,394.597,353.367,173.233,48.159,159.698
C00749=1027.243,394.331,353.414,173.222,48.156,159.696
C00750=1027.233,394.085,353.458,173.212,48.154,159.694
C00751=1027.224,393.840,353.502,173.202,48.152,159.692
C00752=1027.215,393.593,353.544,173.193,48.149,159.690
C00753=1027.205,393.347,353.589,173.182,48.148,159.688
C00754=1027.196,393.102,353.632,173.173,48.145,159.686
C00755=1027.187,392.855,353.675,173.163,48.143,159.684
C00756=1027.176,392.609,353.719,173.153,48.141,159.682
C00757=1027.167,392.364,353.761,173.143,48.139,159.680
C00758=1027.158,392.118,353.805,173.133,48.136,159.678
C00759=1027.148,391.871,353.848,173.124,48.134,159.677
C00760=1027.139,391.626,353.892,173.115,48.132,159.675
C00761=1027.129,391.379,353.935,173.104,48.130,159.673
C00762=1027.120,391.134,353.977,173.095,48.128,159.671
C00763=1027.111,390.887,354.021,173.085,48.126,159.669
C00764=1027.101,390.642,354.063,173.076,48.124,159.667
C00765=1027.092,390.395,354.106,173.066,48.122,159.665
C00766=1027.083,390.149,354.149,173.057,48.119,159.663
C00767=1027.073,389.903,354.193,173.046,48.118,159.661
C00768=1027.064,389.658,354.235,173.037,48.116,159.659
C00769=1027.055,389.411,354.279,173.028,48.114,159.658
C00770=1027.045,389.165,354.321,173.018,48.112,159.656
C00771=1027.036,388.919,354.364,173.009,48.110,159.654
C00772=1027.026,388.673,354.406,172.999,48.108,159.652
C00773=1027.018,388.427,354.449,172.990,48.106,159.650
C00774=1027.008,388.180,354.492,172.981,48.104,159.648
C00775=1026.999,387.934,354.534,172.972,48.102,159.647
C00776=1026.990,387.688,354.576,172.962,48.100,159.645
C00777=1026.981,387.442,354.619,172.953,48.098,159.643
C00778=1026.971,387.196,354.662,172.944,48.097,159.641
C00779=1026.962,386.950,354.705,172.934,48.095,159.639
C00780=1026.953,386.704,354.746,172.925,48.093,159.638
C00781=1026.944,386.458,354.789,172.916,48.091,159.636
C00782=1026.934,386.212,354.832,172.907,48.089,159.634
C00783=1026.925,385.965,354.873,172.897,48.087,159.632
C00784=1026.916,385.719,354.916,172.888,48.086,159.631
C00785=1026.906,385.472,354.958,172.879,48.084,159.629
C00786=1026.897,385.226,354.999,172.870,48.082,159.627
C00787=1026.888,384.980,355.042,172.861,48.081,159.625
C00788=1026.879,384.734,355.084,172.852,48.079,159.624
C00789=1026.870,384.488,355.125,172.842,48.077,159.622
C00790=1026.861,384.242,355.168,172.833,48.075,159.620
C00791=1026.852,383.995,355.209,172.824,48.074,159.619
C00792=1026.843,383.748,355.252,172.816,48.072,159.617
C00793=1026.834,383.502,355.293,172.807,48.070,159.615
C00794=1026.824,383.256,355.336,172.798,48.068,159.613
C00795=1026.816,383.010,355.377,172.789,48.067,159.612
C00796=1026.807,382.763,355.419,172.780,48.065,159.610
C00797=1026.798,382.517,355.461,172.771,48.064,159.609
C00798=1026.789,382.271,355.503,172.763,48.062,159.607
C00799=1026.780,382.024,355.544,172.753,48.061,159.605
C00800=1026.771,381.778,355.586,172.744,48.059,159.604
C00801=1026.763,381.532,355.627,172.735,48.058,159.602
C00802=1026.753,381.294,355.667,172.727,48.056,159.600
C00803=1026.745,381.056,355.708,172.718,48.055,159.599
C00804=1026.736,380.819,355.747,172.710,48.053,159.597
C00805=1026.727,380.581,355.788,172.702,48.052,159.596
C00806=1026.719,380.343,355.828,172.694,48.050,159.594
C00807=1026.710,380.106,355.868,172.685,48.049,159.593
C00808=1026.702,379.868,355.908,172.677,48.047,159.591
C00809=1026.693,379.630,355.948,172.668,48.046,159.590
C00810=1026.685,379.383,355.989,172.660,48.044,159.588
C00811=1026.676,379.137,356.030,172.651,48.043,159.586
C00812=1026.667,378.891,356.072,172.642,48.042,159.585
C00813=1026.659,378.644,356.113,172.634,48.040,159.583
C00814=1026.650,378.398,356.155,172.625,48.039,159.582
C00815=1026.641,378.152,356.196,172.616,48.037,159.580
C00816=1026.633,377.905,356.237,172.608,48.036,159.579
C00817=1026.624,377.659,356.279,172.599,48.034,159.577
C00818=1026.616,377.412,356.319,172.592,48.033,159.576
C00819=1026.607,377.166,356.361,172.583,48.032,159.574
C00820=1026.599,376.920,356.402,172.575,48.030,159.572
C00821=1026.589,376.673,356.442,172.566,48.029,159.571
C00822=1026.581,376.426,356.483,172.557,48.028,159.569
C00823=1026.572,376.181,356.524,172.549,48.026,159.568
C00824=1026.563,375.934,356.565,172.540,48.025,159.566
C00825=1026.555,375.687,356.606,172.533,48.024,159.565
C00826=1026.546,375.441,356.646,172.524,48.023,159.563
C00827=1026.537,375.194,356.687,172.516,48.022,159.562
C00828=1026.528,374.948,356.727,172.507,48.021,159.561
C00829=1026.520,374.701,356.768,172.498,48.019,159.559
C00830=1026.511,374.455,356.808,172.491,48.018,159.558
C00831=1026.502,374.208,356.849,172.482,48.017,159.556
C00832=1026.494,373.962,356.890,172.474,48.016,159.555
C00833=1026.485,373.715,356.930,172.466,48.015,159.553
C00834=1026.477,373.469,356.971,172.458,48.014,159.552
C00835=1026.468,373.222,357.011,172.450,48.012,159.551
C00836=1026.460,372.976,357.052,172.441,48.011,159.549
C00837=1026.451,372.729,357.093,172.434,48.010,159.548
C00838=1026.442,372.482,357.132,172.425,48.009,159.546
C00839=1026.434,372.236,357.173,172.417,48.008,159.545
C00840=1026.425,371.989,357.213,172.408,48.007,159.543
C00841=1026.417,371.743,357.254,172.401,48.006,159.542
C00842=1026.409,371.496,357.293,172.393,48.005,159.541
C00843=1026.400,371.249,357.334,172.385,48.004,159.539
C00844=1026.392,371.003,357.375,172.377,48.003,159.538
C00845=1026.383,370.756,357.414,172.368,48.002,159.536
C00846=1026.375,370.509,357.455,172.361,48.001,159.535
C00847=1026.366,370.263,357.494,172.353,47.999,159.534
C00848=1026.358,370.017,357.535,172.345,47.999,159.532
C00849=1026.351,369.770,357.575,172.337,47.998,159.531
C00850=1026.342,369.524,357.615,172.329,47.997,159.530
C00851=1026.334,369.276,357.655,172.322,47.995,159.528
C00852=1026.325,369.030,357.695,172.313,47.995,159.527
C00853=1026.317,368.783,357.735,172.306,47.994,159.526
C00854=1026.309,368.537,357.774,172.298,47.993,159.524
C00855=1026.300,368.291,357.815,172.289,47.992,159.523
C00856=1026.292,368.043,357.855,172.282,47.991,159.522
C00857=1026.283,367.796,357.894,172.274,47.990,159.521
C00858=1026.275,367.550,357.933,172.266,47.989,159.519
C00859=1026.266,367.303,357.973,172.258,47.989,159.518
C00860=1026.258,367.056,358.013,172.251,47.988,159.517
C00861=1026.250,366.810,358.052,172.243,47.987,159.515
C00862=1026.242,366.582,358.089,172.236,47.986,159.514
C00863=1026.234,366.356,358.125,172.229,47.986,159.513
C00864=1026.227,366.129,358.161,172.221,47.985,159.512
C00865=1026.219,365.901,358.198,172.215,47.984,159.511
C00866=1026.211,365.674,358.233,172.208,47.984,159.510
C00867=1026.204,365.447,358.270,172.200,47.983,159.508
C00868=1026.197,365.220,358.307,172.193,47.982,159.507
C00869=1026.188,364.993,358.343,172.187,47.981,159.506
C00870=1026.180,364.746,358.383,172.179,47.981,159.505
C00871=1026.172,364.499,358.421,172.171,47.980,159.504
C00872=1026.164,364.253,358.460,172.164,47.980,159.502
C00873=1026.156,364.006,358.500,172.156,47.979,159.501
C00874=1026.148,363.759,358.540,172.149,47.978,159.500
C00875=1026.140,363.512,358.578,172.141,47.977,159.499
C00876=1026.132,363.265,358.618,172.134,47.977,159.498
C00877=1026.123,363.019,358.657,172.125,47.976,159.496
C00878=1026.115,362.772,358.696,172.118,47.976,159.495
C00879=1026.107,362.525,358.735,172.111,47.975,159.494
C00880=1026.099,362.279,358.774,172.103,47.974,159.493
C00881=1026.091,362.032,358.813,172.096,47.974,159.492
C00882=1026.083,361.785,358.852,172.089,47.973,159.490
C00883=1026.075,361.538,358.892,172.081,47.972,159.489
C00884=1026.067,361.291,358.931,172.074,47.972,159.488
C00885=1026.059,361.044,358.969,172.067,47.972,159.487
C00886=1026.051,360.798,359.008,172.060,47.971,159.486
C00887=1026.043,360.551,359.047,172.052,47.970,159.485
C00888=1026.035,360.303,359.086,172.045,47.970,159.483
C00889=1026.028,360.057,359.125,172.037,47.969,159.482
C00890=1026.019,359.810,359.164,172.030,47.969,159.481
C00891=1026.011,359.563,359.202,172.022,47.969,159.480
C00892=1026.003,359.316,359.241,172.015,47.968,159.479
C00893=1025.994,359.070,359.279,172.008,47.968,159.478
C00894=1025.986,358.823,359.318,172.000,47.967,159.477
C00895=1025.978,358.576,359.357,171.993,47.967,159.476
C00896=1025.971,358.329,359.395,171.986,47.967,159.475
C00897=1025.962,358.082,359.433,171.979,47.966,159.473
C00898=1025.955,357.835,359.472,171.972,47.966,159.472
C00899=1025.947,357.588,359.510,171.964,47.965,159.471
C00900=1025.939,357.341,359.549,171.957,47.965,159.470
C00901=1025.931,357.094,359.587,171.950,47.965,159.469
C00902=1025.923,356.847,359.626,171.943,47.965,159.468
C00903=1025.915,356.601,359.664,171.936,47.964,159.467
C00904=1025.907,356.353,359.703,171.929,47.964,159.466
C00905=1025.899,356.107,359.740,171.921,47.963,159.465
C00906=1025.891,355.859,359.778,171.914,47.963,159.464
C00907=1025.884,355.613,359.816,171.908,47.963,159.463
C00908=1025.875,355.366,359.855,171.901,47.962,159.462
C00909=1025.868,355.119,359.893,171.894,47.962,159.461
C00910=1025.860,354.872,359.932,171.887,47.962,159.460
C00911=1025.852,354.625,359.969,171.879,47.961,159.458
C00912=1025.844,354.378,360.007,171.872,47.961,159.457
C00913=1025.836,354.131,360.046,171.865,47.961,159.457
C00914=1025.828,353.883,360.084,171.858,47.961,159.456
C00915=1025.821,353.637,360.122,171.851,47.961,159.455
C00916=1025.812,353.389,360.159,171.844,47.960,159.453
C00917=1025.804,353.143,360.197,171.837,47.960,159.452
C00918=1025.797,352.896,360.235,171.830,47.960,159.451
C00919=1025.788,352.649,360.273,171.824,47.960,159.450
C00920=1025.781,352.402,360.310,171.817,47.960,159.449
C00921=1025.773,352.155,360.349,171.810,47.960,159.448
C00922=1025.766,351.931,360.383,171.804,47.960,159.448
C00923=1025.759,351.707,360.417,171.797,47.959,159.447
C00924=1025.752,351.483,360.451,171.791,47.960,159.446
C00925=1025.745,351.259,360.485,171.785,47.959,159.445
C00926=1025.738,351.035,360.519,171.778,47.959,159.444
C00927=1025.730,350.812,360.553,171.772,47.960,159.443
C00928=1025.724,350.588,360.588,171.766,47.959,159.442
C00929=1025.717,350.364,360.622,171.760,47.959,159.441
C00930=1025.709,350.117,360.659,171.754,47.959,159.441
C00931=1025.701,349.870,360.696,171.747,47.959,159.440
C00932=1025.694,349.623,360.734,171.740,47.959,159.439
C00933=1025.686,349.376,360.772,171.733,47.959,159.438
C00934=1025.678,349.129,360.809,171.727,47.959,159.437
C00935=1025.671,348.882,360.847,171.720,47.959,159.436
C00936=1025.664,348.635,360.884,171.713,47.959,159.435
C00937=1025.656,348.388,360.921,171.706,47.959,159.434
C00938=1025.648,348.141,360.959,171.700,47.959,159.433
C00939=1025.641,347.893,360.997,171.693,47.959,159.432
C00940=1025.633,347.646,361.034,171.686,47.959,159.431
C00941=1025.625,347.399,361.071,171.679,47.959,159.430
C00942=1025.617,347.152,361.108,171.673,47.960,159.429
C00943=1025.609,346.905,361.145,171.666,47.959,159.429
C00944=1025.602,346.658,361.182,171.659,47.959,159.428
C00945=1025.594,346.411,361.219,171.653,47.960,159.427
C00946=1025.587,346.164,361.256,171.647,47.960,159.426
C00947=1025.579,345.917,361.293,171.640,47.960,159.425
C00948=1025.571,345.669,361.331,171.633,47.960,159.424
C00949=1025.564,345.422,361.367,171.626,47.961,159.423
C00950=1025.556,345.175,361.404,171.620,47.960,159.422
C00951=1025.548,344.928,361.442,171.614,47.961,159.422
C00952=1025.541,344.680,361.478,171.607,47.961,159.421
C00953=1025.534,344.433,361.516,171.601,47.961,159.420
C00954=1025.526,344.186,361.552,171.594,47.962,159.419
C00955=1025.518,343.939,361.589,171.587,47.961,159.418
C00956=1025.511,343.692,361.626,171.582,47.962,159.417
C00957=1025.504,343.445,361.662,171.575,47.962,159.417
C00958=1025.496,343.198,361.699,171.568,47.962,159.416
C00959=1025.489,342.950,361.736,171.561,47.963,159.415
C00960=1025.481,342.703,361.773,171.555,47.963,159.414
C00961=1025.474,342.456,361.810,171.548,47.963,159.413
C00962=1025.466,342.209,361.846,171.543,47.963,159.412
C00963=1025.458,341.961,361.883,171.536,47.964,159.412
C00964=1025.451,341.714,361.920,171.529,47.964,159.411
C00965=1025.443,341.467,361.956,171.524,47.964,159.410
C00966=1025.436,341.220,361.992,171.517,47.964,159.409
C00967=1025.428,340.973,362.029,171.510,47.965,159.408
C00968=1025.421,340.726,362.066,171.504,47.965,159.407
C00969=1025.413,340.478,362.102,171.498,47.966,159.407
C00970=1025.406,340.231,362.138,171.492,47.966,159.406
C00971=1025.399,339.984,362.176,171.485,47.966,159.405
C00972=1025.391,339.737,362.212,171.478,47.967,159.404
C00973=1025.384,339.489,362.248,171.473,47.967,159.404
C00974=1025.376,339.242,362.284,171.466,47.968,159.403
C00975=1025.368,338.994,362.320,171.460,47.968,159.402
C00976=1025.361,338.748,362.356,171.454,47.969,159.401
C00977=1025.354,338.500,362.393,171.447,47.969,159.400
C00978=1025.346,338.253,362.429,171.441,47.969,159.400
C00979=1025.339,338.006,362.465,171.435,47.970,159.399
C00980=1025.331,337.759,362.501,171.429,47.970,159.398
C00981=1025.324,337.511,362.537,171.422,47.971,159.397
C00982=1025.317,337.286,362.570,171.417,47.972,159.397
C00983=1025.310,337.061,362.604,171.411,47.972,159.396
C00984=1025.304,336.835,362.636,171.406,47.972,159.395
C00985=1025.297,336.610,362.669,171.400,47.973,159.395
C00986=1025.290,336.385,362.702,171.394,47.973,159.394
C00987=1025.284,336.159,362.735,171.389,47.974,159.394
C00988=1025.277,335.933,362.767,171.383,47.974,159.393
C00989=1025.270,335.708,362.800,171.378,47.974,159.392
C00990=1025.263,335.461,362.836,171.371,47.976,159.392
C00991=1025.255,335.214,362.872,171.366,47.976,159.391
C00992=1025.248,334.967,362.908,171.359,47.976,159.390
C00993=1025.241,334.719,362.944,171.353,47.978,159.389
C00994=1025.234,334.471,362.980,171.347,47.978,159.389
C00995=1025.227,334.224,363.016,171.340,47.978,159.388
C00996=1025.219,333.976,363.051,171.335,47.979,159.387
C00997=1025.212,333.730,363.087,171.328,47.980,159.387
C00998=1025.205,333.482,363.124,171.323,47.980,159.386
C00999=1025.198,333.235,363.159,171.316,47.981,159.385
C01000=1025.189,332.988,363.194,171.310,47.981,159.384
C01001=1025.183,332.740,363.229,171.304,47.982,159.384
C01002=1025.175,332.493,363.266,171.299,47.983,159.383
C01003=1025.168,332.245,363.301,171.292,47.984,159.383
C01004=1025.161,331.997,363.336,171.287,47.985,159.382
C01005=1025.153,331.751,363.372,171.281,47.985,159.381
C01006=1025.146,331.504,363.407,171.275,47.986,159.381
C01007=1025.139,331.256,363.443,171.269,47.986,159.380
C01008=1025.132,331.009,363.478,171.263,47.988,159.379
C01009=1025.124,330.761,363.513,171.257,47.988,159.379
C01010=1025.117,330.514,363.549,171.251,47.989,159.378
C01011=1025.109,330.266,363.584,171.245,47.990,159.377
C01012=1025.102,330.019,363.619,171.239,47.991,159.377
C01013=1025.096,329.771,363.655,171.233,47.991,159.376
C01014=1025.088,329.524,363.691,171.227,47.992,159.375
C01015=1025.081,329.277,363.725,171.221,47.993,159.375
C01016=1025.074,329.030,363.760,171.216,47.994,159.374
C01017=1025.066,328.782,363.796,171.209,47.995,159.374
C01018=1025.060,328.534,363.831,171.204,47.995,159.373
C01019=1025.053,328.287,363.867,171.198,47.997,159.372
C01020=1025.045,328.040,363.901,171.192,47.997,159.372
C01021=1025.038,327.792,363.937,171.186,47.998,159.371
C01022=1025.031,327.545,363.972,171.180,47.999,159.371
C01023=1025.024,327.298,364.007,171.175,48.000,159.370
C01024=1025.016,327.050,364.042,171.168,48.001,159.369
C01025=1025.009,326.802,364.077,171.163,48.002,159.369
C01026=1025.002,326.555,364.112,171.157,48.003,159.368
C01027=1024.995,326.308,364.146,171.151,48.004,159.368
C01028=1024.987,326.060,364.181,171.145,48.005,159.367
C01029=1024.980,325.813,364.216,171.140,48.006,159.367
C01030=1024.972,325.566,364.250,171.134,48.007,159.366
C01031=1024.965,325.318,364.285,171.128,48.008,159.365
C01032=1024.958,325.070,364.320,171.123,48.009,159.365
C01033=1024.950,324.823,364.354,171.116,48.010,159.364
C01034=1024.943,324.575,364.389,171.111,48.011,159.364
C01035=1024.936,324.328,364.423,171.106,48.012,159.363
C01036=1024.929,324.080,364.458,171.099,48.013,159.363
C01037=1024.921,323.833,364.493,171.094,48.014,159.362
C01038=1024.914,323.585,364.527,171.088,48.016,159.362
C01039=1024.907,323.338,364.562,171.083,48.017,159.361
C01040=1024.900,323.091,364.597,171.077,48.018,159.361
C01041=1024.893,322.843,364.630,171.071,48.019,159.360
C01042=1024.886,322.615,364.662,171.066,48.020,159.360
C01043=1024.880,322.388,364.694,171.060,48.021,159.359
C01044=1024.873,322.160,364.726,171.055,48.022,159.359
C01045=1024.867,321.933,364.758,171.050,48.023,159.358
C01046=1024.859,321.705,364.788,171.046,48.024,159.358
C01047=1024.853,321.477,364.821,171.040,48.025,159.357
C01048=1024.847,321.249,364.852,171.035,48.026,159.357
C01049=1024.840,321.022,364.884,171.030,48.027,159.356
C01050=1024.833,320.774,364.918,171.024,48.028,159.356
C01051=1024.826,320.527,364.953,171.019,48.030,159.355
C01052=1024.819,320.279,364.987,171.013,48.031,159.355
C01053=1024.811,320.032,365.022,171.007,48.032,159.354
C01054=1024.805,319.784,365.056,171.002,48.033,159.354
C01055=1024.797,319.536,365.090,170.996,48.034,159.353
C01056=1024.791,319.290,365.124,170.991,48.036,159.353
C01057=1024.784,319.042,365.158,170.985,48.037,159.352
C01058=1024.777,318.794,365.192,170.980,48.038,159.352
C01059=1024.769,318.547,365.227,170.975,48.039,159.351
C01060=1024.763,318.299,365.261,170.969,48.041,159.351
C01061=1024.756,318.051,365.295,170.963,48.042,159.351
C01062=1024.748,317.804,365.329,170.958,48.043,159.350
C01063=1024.741,317.556,365.363,170.952,48.044,159.350
C01064=1024.735,317.309,365.398,170.947,48.046,159.349
C01065=1024.727,317.061,365.432,170.941,48.047,159.349
C01066=1024.721,316.814,365.465,170.936,48.048,159.348
C01067=1024.714,316.566,365.499,170.930,48.049,159.348
C01068=1024.707,316.318,365.533,170.925,48.051,159.347
C01069=1024.700,316.071,365.567,170.920,48.052,159.347
C01070=1024.693,315.823,365.602,170.915,48.053,159.346
C01071=1024.686,315.576,365.636,170.909,48.055,159.346
C01072=1024.679,315.329,365.670,170.903,48.056,159.345
C01073=1024.673,315.081,365.704,170.898,48.057,159.345
C01074=1024.666,314.833,365.738,170.893,48.059,159.345
C01075=1024.659,314.586,365.771,170.887,48.060,159.344
C01076=1024.652,314.338,365.805,170.882,48.061,159.344
C01077=1024.645,314.090,365.839,170.877,48.063,159.343
C01078=1024.638,313.843,365.873,170.871,48.064,159.343
C01079=1024.632,313.596,365.907,170.866,48.065,159.342
C01080=1024.625,313.348,365.941,170.860,48.067,159.342
C01081=1024.618,313.100,365.975,170.855,48.068,159.342
C01082=1024.611,312.853,366.008,170.850,48.069,159.341
C01083=1024.605,312.605,366.042,170.845,48.071,159.341
C01084=1024.598,312.357,366.076,170.840,48.072,159.340
C01085=1024.591,312.110,366.109,170.834,48.074,159.340
C01086=1024.584,311.862,366.143,170.829,48.075,159.340
C01087=1024.578,311.615,366.177,170.823,48.076,159.339
C01088=1024.571,311.367,366.211,170.818,48.078,159.339
C01089=1024.564,311.120,366.245,170.813,48.079,159.338
C01090=1024.558,310.872,366.278,170.808,48.081,159.338
C01091=1024.551,310.624,366.312,170.802,48.083,159.338
C01092=1024.545,310.377,366.346,170.797,48.084,159.337
C01093=1024.537,310.129,366.378,170.792,48.085,159.337
C01094=1024.530,309.882,366.412,170.787,48.087,159.336
C01095=1024.523,309.634,366.445,170.781,48.089,159.336
C01096=1024.515,309.386,366.478,170.776,48.090,159.336
C01097=1024.509,309.139,366.511,170.771,48.092,159.335
C01098=1024.502,308.891,366.544,170.766,48.094,159.335
C01099=1024.494,308.643,366.577,170.760,48.096,159.335
C01100=1024.488,308.396,366.610,170.755,48.097,159.334
C01101=1024.481,308.148,366.644,170.750,48.099,159.334
C01102=1024.474,307.923,366.673,170.745,48.100,159.334
C01103=1024.468,307.698,366.703,170.740,48.102,159.333
C01104=1024.462,307.473,366.733,170.736,48.103,159.333
C01105=1024.456,307.247,366.763,170.731,48.105,159.333
C01106=1024.449,307.022,366.793,170.726,48.106,159.332
C01107=1024.443,306.797,366.823,170.721,48.108,159.332
C01108=1024.436,306.572,366.853,170.718,48.110,159.332
C01109=1024.430,306.348,366.882,170.712,48.111,159.332
C01110=1024.423,306.100,366.916,170.707,48.113,159.331
C01111=1024.417,305.852,366.948,170.703,48.115,159.331
C01112=1024.409,305.604,366.981,170.697,48.117,159.331
C01113=1024.403,305.357,367.014,170.692,48.118,159.330
C01114=1024.396,305.109,367.047,170.687,48.120,159.330
C01115=1024.389,304.862,367.079,170.682,48.122,159.330
C01116=1024.382,304.613,367.113,170.677,48.123,159.329
C01117=1024.375,304.366,367.145,170.671,48.126,159.329
C01118=1024.368,304.118,367.178,170.666,48.127,159.329
C01119=1024.362,303.870,367.211,170.661,48.129,159.329
C01120=1024.355,303.623,367.243,170.656,48.131,159.328
C01121=1024.348,303.375,367.276,170.651,48.132,159.328
C01122=1024.341,303.128,367.309,170.647,48.134,159.328
C01123=1024.334,302.880,367.341,170.642,48.136,159.327
C01124=1024.327,302.632,367.375,170.636,48.138,159.327
C01125=1024.321,302.384,367.407,170.631,48.140,159.327
C01126=1024.313,302.136,367.440,170.626,48.142,159.327
C01127=1024.307,301.889,367.473,170.621,48.143,159.326
C01128=1024.301,301.641,367.505,170.616,48.145,159.326
C01129=1024.294,301.393,367.537,170.611,48.147,159.326
C01130=1024.287,301.145,367.570,170.607,48.149,159.325
C01131=1024.280,300.898,367.602,170.601,48.151,159.325
C01132=1024.274,300.650,367.635,170.596,48.153,159.325
C01133=1024.267,300.402,367.668,170.591,48.154,159.325
C01134=1024.260,300.155,367.700,170.586,48.156,159.324
C01135=1024.254,299.907,367.733,170.581,48.159,159.324
C01136=1024.247,299.659,367.765,170.576,48.160,159.324
C01137=1024.240,299.411,367.797,170.572,48.162,159.324
C01138=1024.234,299.163,367.830,170.567,48.164,159.323
C01139=1024.227,298.916,367.862,170.562,48.166,159.323
C01140=1024.220,298.668,367.895,170.556,48.168,159.323
C01141=1024.214,298.421,367.928,170.551,48.170,159.322
C01142=1024.207,298.172,367.959,170.546,48.172,159.322
C01143=1024.201,297.925,367.992,170.542,48.174,159.322
C01144=1024.194,297.677,368.025,170.537,48.175,159.322
C01145=1024.188,297.429,368.056,170.532,48.178,159.322
C01146=1024.181,297.181,368.089,170.527,48.180,159.321
C01147=1024.174,296.934,368.121,170.523,48.182,159.321
C01148=1024.168,296.685,368.154,170.518,48.183,159.321
C01149=1024.161,296.438,368.186,170.513,48.185,159.321
C01150=1024.154,296.190,368.219,170.508,48.188,159.320
C01151=1024.148,295.942,368.251,170.503,48.190,159.320
C01152=1024.142,295.695,368.283,170.498,48.191,159.320
C01153=1024.135,295.447,368.315,170.494,48.193,159.320
C01154=1024.129,295.199,368.347,170.489,48.195,159.320
C01155=1024.122,294.952,368.380,170.483,48.198,159.319
C01156=1024.116,294.704,368.412,170.478,48.199,159.319
C01157=1024.110,294.456,368.444,170.473,48.201,159.319
C01158=1024.103,294.208,368.476,170.469,48.204,159.319
C01159=1024.097,293.960,368.509,170.464,48.206,159.318
C01160=1024.089,293.712,368.540,170.459,48.208,159.318
C01161=1024.083,293.464,368.572,170.455,48.210,159.318
C01162=1024.078,293.248,368.600,170.451,48.212,159.318
C01163=1024.072,293.031,368.628,170.446,48.214,159.318
C01164=1024.065,292.815,368.656,170.443,48.216,159.318
C01165=1024.060,292.599,368.683,170.438,48.217,159.317
C01166=1024.054,292.383,368.711,170.434,48.219,159.317
C01167=1024.048,292.166,368.739,170.430,48.221,159.317
C01168=1024.043,291.949,368.767,170.425,48.223,159.317
C01169=1024.037,291.733,368.794,170.422,48.225,159.317
C01170=1024.030,291.485,368.826,170.417,48.227,159.317
C01171=1024.023,291.238,368.858,170.412,48.229,159.316
C01172=1024.017,290.990,368.890,170.408,48.232,159.316
C01173=1024.010,290.742,368.921,170.402,48.234,159.316
C01174=1024.004,290.494,368.953,170.397,48.236,159.316
C01175=1023.997,290.246,368.984,170.393,48.239,159.316
C01176=1023.990,289.998,369.016,170.388,48.241,159.316
C01177=1023.983,289.750,369.047,170.383,48.243,159.315
C01178=1023.977,289.502,369.078,170.379,48.246,159.315
C01179=1023.971,289.254,369.110,170.374,48.248,159.315
C01180=1023.964,289.006,369.142,170.370,48.250,159.315
C01181=1023.957,288.758,369.173,170.365,48.252,159.315
C01182=1023.951,288.510,369.205,170.360,48.255,159.315
C01183=1023.944,288.262,369.236,170.356,48.257,159.315
C01184=1023.937,288.014,369.268,170.351,48.259,159.315
C01185=1023.930,287.767,369.299,170.346,48.261,159.314
C01186=1023.924,287.519,369.330,170.342,48.264,159.314
C01187=1023.918,287.271,369.362,170.337,48.266,159.314
C01188=1023.911,287.024,369.393,170.333,48.268,159.314
C01189=1023.904,286.776,369.424,170.328,48.271,159.314
C01190=1023.898,286.527,369.456,170.323,48.273,159.314
C01191=1023.892,286.279,369.487,170.318,48.276,159.314
C01192=1023.885,286.031,369.519,170.313,48.278,159.314
C01193=1023.878,285.783,369.550,170.309,48.281,159.313
C01194=1023.872,285.536,369.581,170.304,48.283,159.313
C01195=1023.865,285.288,369.612,170.300,48.285,159.313
C01196=1023.859,285.039,369.643,170.295,48.288,159.313
C01197=1023.852,284.792,369.674,170.291,48.290,159.313
C01198=1023.845,284.544,369.705,170.286,48.293,159.313
C01199=1023.838,284.295,369.736,170.281,48.295,159.313
C01200=1023.832,284.048,369.767,170.277,48.298,159.313
C01201=1023.826,283.800,369.799,170.272,48.300,159.313
C01202=1023.819,283.552,369.829,170.268,48.303,159.313
C01203=1023.812,283.304,369.860,170.263,48.305,159.312
C01204=1023.805,283.056,369.891,170.259,48.308,159.312
C01205=1023.799,282.809,369.922,170.254,48.310,159.312
C01206=1023.793,282.560,369.953,170.250,48.313,159.312
C01207=1023.786,282.312,369.984,170.245,48.316,159.312
C01208=1023.779,282.064,370.014,170.241,48.318,159.312
C01209=1023.772,281.816,370.046,170.236,48.321,159.312
C01210=1023.766,281.568,370.076,170.232,48.323,159.312
C01211=1023.760,281.320,370.108,170.227,48.325,159.312
C01212=1023.753,281.072,370.138,170.223,48.328,159.312
C01213=1023.747,280.825,370.169,170.218,48.331,159.312
C01214=1023.740,280.576,370.199,170.214,48.333,159.312
C01215=1023.733,280.328,370.231,170.209,48.336,159.312
C01216=1023.727,280.080,370.262,170.205,48.339,159.312
C01217=1023.721,279.833,370.293,170.200,48.341,159.312
C01218=1023.714,279.584,370.323,170.196,48.344,159.312
C01219=1023.708,279.336,370.354,170.192,48.346,159.312
C01220=1023.701,279.089,370.385,170.187,48.349,159.311
C01221=1023.694,278.840,370.415,170.182,48.351,159.311
C01222=1023.690,278.630,370.441,170.178,48.354,159.311
C01223=1023.684,278.420,370.468,170.174,48.356,159.311
C01224=1023.679,278.209,370.493,170.171,48.358,159.311
C01225=1023.673,277.999,370.519,170.167,48.360,159.311
C01226=1023.667,277.789,370.545,170.163,48.363,159.311
C01227=1023.662,277.578,370.571,170.159,48.365,159.311
C01228=1023.657,277.368,370.597,170.156,48.367,159.311
C01229=1023.651,277.158,370.624,170.152,48.369,159.311
C01230=1023.645,276.910,370.654,170.148,48.372,159.311
C01231=1023.638,276.662,370.684,170.143,48.375,159.311
C01232=1023.632,276.414,370.715,170.139,48.378,159.311
C01233=1023.625,276.166,370.745,170.135,48.380,159.311
C01234=1023.618,275.917,370.775,170.130,48.383,159.311
C01235=1023.612,275.670,370.806,170.126,48.386,159.311
C01236=1023.605,275.422,370.837,170.122,48.389,159.311
C01237=1023.599,275.174,370.866,170.117,48.392,159.311
C01238=1023.592,274.926,370.897,170.113,48.394,159.311
C01239=1023.586,274.677,370.928,170.108,48.397,159.311
C01240=1023.579,274.430,370.958,170.104,48.400,159.311
C01241=1023.573,274.181,370.988,170.100,48.403,159.311
C01242=1023.566,273.934,371.018,170.095,48.406,159.311
C01243=1023.560,273.685,371.049,170.091,48.408,159.311
C01244=1023.553,273.438,371.079,170.087,48.411,159.311
C01245=1023.547,273.189,371.109,170.082,48.414,159.311
C01246=1023.540,272.942,371.139,170.078,48.417,159.311
C01247=1023.534,272.693,371.170,170.073,48.420,159.311
C01248=1023.528,272.445,371.199,170.069,48.422,159.311
C01249=1023.521,272.197,371.230,170.065,48.425,159.311
C01250=1023.515,271.949,371.259,170.060,48.428,159.311
C01251=1023.508,271.701,371.290,170.056,48.431,159.311
C01252=1023.502,271.453,371.320,170.052,48.434,159.311
C01253=1023.495,271.204,371.350,170.048,48.437,159.311
C01254=1023.489,270.956,371.380,170.043,48.440,159.311
C01255=1023.483,270.708,371.410,170.039,48.443,159.311
C01256=1023.476,270.460,371.440,170.034,48.445,159.311
C01257=1023.470,270.212,371.471,170.030,48.449,159.311
C01258=1023.463,269.964,371.500,170.026,48.452,159.311
C01259=1023.457,269.716,371.529,170.022,48.454,159.311
C01260=1023.450,269.468,371.560,170.017,48.457,159.311
C01261=1023.444,269.220,371.590,170.013,48.461,159.311
C01262=1023.437,268.971,371.619,170.009,48.463,159.311
C01263=1023.431,268.723,371.650,170.005,48.466,159.311
C01264=1023.425,268.476,371.679,170.000,48.470,159.312
C01265=1023.418,268.227,371.709,169.996,48.473,159.312
C01266=1023.412,267.979,371.739,169.992,48.475,159.312
C01267=1023.405,267.730,371.769,169.988,48.479,159.312
C01268=1023.399,267.483,371.798,169.983,48.482,159.312
C01269=1023.393,267.235,371.829,169.979,48.484,159.312
C01270=1023.386,266.986,371.858,169.975,48.488,159.312
C01271=1023.379,266.739,371.888,169.971,48.491,159.312
C01272=1023.373,266.490,371.917,169.966,48.493,159.312
C01273=1023.367,266.242,371.948,169.962,48.497,159.312
C01274=1023.360,265.994,371.977,169.958,48.500,159.312
C01275=1023.353,265.746,372.007,169.954,48.503,159.312
C01276=1023.347,265.498,372.036,169.949,48.506,159.312
C01277=1023.341,265.250,372.065,169.945,48.509,159.313
C01278=1023.334,265.001,372.096,169.941,48.512,159.312
C01279=1023.328,264.753,372.125,169.937,48.516,159.313
C01280=1023.322,264.505,372.154,169.933,48.518,159.313
C01281=1023.315,264.257,372.183,169.929,48.522,159.313
C01282=1023.304,263.841,372.233,169.921,48.527,159.313
C01283=1023.294,263.424,372.283,169.914,48.532,159.313
C01284=1023.283,263.009,372.332,169.908,48.538,159.313
C01285=1023.272,262.593,372.381,169.900,48.543,159.313
C01286=1023.266,262.345,372.411,169.896,48.546,159.313
C01287=1023.259,262.097,372.440,169.892,48.550,159.314
C01288=1023.252,261.848,372.469,169.888,48.553,159.314
C01289=1023.247,261.600,372.499,169.883,48.556,159.314
C01290=1023.240,261.352,372.528,169.879,48.559,159.314
C01291=1023.234,261.104,372.557,169.876,48.562,159.314
C01292=1023.227,260.855,372.587,169.872,48.565,159.314
C01293=1023.221,260.607,372.616,169.868,48.569,159.314
C01294=1023.215,260.359,372.645,169.864,48.572,159.315
C01295=1023.209,260.111,372.674,169.859,48.575,159.315
C01296=1023.202,259.863,372.702,169.854,48.579,159.315
C01297=1023.195,259.615,372.731,169.850,48.582,159.315
C01298=1023.188,259.366,372.761,169.846,48.586,159.315
C01299=1023.182,259.118,372.790,169.842,48.589,159.315
C01300=1023.175,258.870,372.818,169.838,48.593,159.315
C01301=1023.169,258.622,372.847,169.834,48.596,159.316
C01302=1023.162,258.373,372.877,169.830,48.600,159.316
C01303=1023.155,258.125,372.905,169.826,48.602,159.316
C01304=1023.149,257.877,372.934,169.822,48.606,159.316
C01305=1023.143,257.629,372.963,169.818,48.609,159.316
C01306=1023.136,257.381,372.992,169.814,48.613,159.316
C01307=1023.129,257.132,373.020,169.810,48.616,159.316
C01308=1023.123,256.884,373.050,169.806,48.620,159.317
C01309=1023.117,256.636,373.079,169.802,48.623,159.317
C01310=1023.110,256.387,373.108,169.798,48.627,159.317
C01311=1023.103,256.140,373.136,169.793,48.630,159.317
C01312=1023.097,255.891,373.164,169.789,48.634,159.317
C01313=1023.091,255.643,373.193,169.785,48.637,159.317
C01314=1023.084,255.394,373.222,169.781,48.641,159.318
C01315=1023.077,255.146,373.251,169.777,48.644,159.318
C01316=1023.071,254.898,373.280,169.773,48.648,159.318
C01317=1023.065,254.649,373.309,169.769,48.651,159.318
C01318=1023.058,254.401,373.337,169.765,48.654,159.318
C01319=1023.052,254.153,373.366,169.761,48.658,159.318
C01320=1023.046,253.904,373.394,169.757,48.661,159.319
C01321=1023.039,253.657,373.423,169.753,48.665,159.319
C01322=1023.033,253.409,373.452,169.749,48.668,159.319
C01323=1023.026,253.160,373.481,169.745,48.672,159.319
C01324=1023.020,252.912,373.509,169.741,48.675,159.319
C01325=1023.014,252.664,373.538,169.737,48.679,159.320
C01326=1023.008,252.415,373.566,169.733,48.683,159.320
C01327=1023.001,252.167,373.595,169.729,48.686,159.320
C01328=1022.994,251.919,373.624,169.725,48.690,159.320
C01329=1022.988,251.670,373.652,169.721,48.693,159.320
C01330=1022.982,251.422,373.681,169.717,48.697,159.321
C01331=1022.975,251.174,373.709,169.713,48.700,159.321
C01332=1022.969,250.926,373.738,169.709,48.704,159.321
C01333=1022.963,250.678,373.767,169.706,48.708,159.321
C01334=1022.956,250.429,373.794,169.702,48.711,159.321
C01335=1022.950,250.181,373.823,169.698,48.715,159.322
C01336=1022.944,249.932,373.852,169.694,48.718,159.322
C01337=1022.938,249.684,373.881,169.689,48.722,159.322
C01338=1022.927,249.266,373.928,169.683,48.728,159.322
C01339=1022.917,248.849,373.977,169.676,48.734,159.323
C01340=1022.905,248.431,374.024,169.670,48.740,159.323
C01341=1022.895,248.013,374.073,169.663,48.747,159.323
C01342=1022.888,247.765,374.100,169.659,48.750,159.324
C01343=1022.883,247.518,374.129,169.655,48.754,159.324
C01344=1022.877,247.269,374.157,169.651,48.758,159.324
C01345=1022.870,247.020,374.185,169.648,48.761,159.324
C01346=1022.864,246.772,374.214,169.644,48.764,159.325
C01347=1022.858,246.523,374.242,169.640,48.769,159.325
C01348=1022.851,246.276,374.271,169.636,48.772,159.325
C01349=1022.845,246.027,374.299,169.632,48.776,159.325
C01350=1022.840,245.779,374.327,169.628,48.779,159.325
C01351=1022.833,245.531,374.356,169.624,48.783,159.326
C01352=1022.827,245.282,374.384,169.620,48.787,159.326
C01353=1022.821,245.034,374.412,169.616,48.790,159.326
C01354=1022.814,244.786,374.441,169.613,48.794,159.326
C01355=1022.808,244.537,374.469,169.609,48.798,159.327
C01356=1022.803,244.289,374.497,169.605,48.801,159.327
C01357=1022.796,244.040,374.525,169.601,48.806,159.327
C01358=1022.790,243.792,374.554,169.597,48.809,159.327
C01359=1022.784,243.544,374.582,169.593,48.813,159.328
C01360=1022.777,243.295,374.610,169.589,48.817,159.328
C01361=1022.771,243.047,374.637,169.586,48.821,159.328
C01362=1022.765,242.799,374.665,169.582,48.824,159.328
C01363=1022.758,242.550,374.693,169.578,48.828,159.329
C01364=1022.752,242.302,374.722,169.574,48.832,159.329
C01365=1022.745,242.054,374.750,169.570,48.836,159.329
C01366=1022.739,241.806,374.777,169.566,48.840,159.329
C01367=1022.733,241.557,374.806,169.563,48.844,159.330
C01368=1022.727,241.309,374.833,169.559,48.848,159.330
C01369=1022.721,241.060,374.862,169.555,48.851,159.330
C01370=1022.715,240.812,374.889,169.551,48.856,159.331
C01371=1022.708,240.564,374.917,169.547,48.859,159.331
C01372=1022.702,240.315,374.945,169.544,48.863,159.331
C01373=1022.695,240.067,374.973,169.540,48.867,159.331
C01374=1022.690,239.819,375.001,169.536,48.871,159.332
C01375=1022.683,239.570,375.029,169.532,48.875,159.332
C01376=1022.677,239.322,375.056,169.528,48.879,159.332
C01377=1022.670,239.073,375.084,169.524,48.883,159.333
C01378=1022.664,238.825,375.111,169.521,48.887,159.333
C01379=1022.658,238.576,375.139,169.517,48.891,159.333
C01380=1022.652,238.328,375.167,169.513,48.895,159.333
C01381=1022.645,238.079,375.194,169.509,48.899,159.334
C01382=1022.639,237.831,375.222,169.506,48.903,159.334
C01383=1022.632,237.583,375.250,169.502,48.907,159.335
C01384=1022.626,237.334,375.277,169.498,48.911,159.335
C01385=1022.620,237.086,375.304,169.494,48.915,159.335
C01386=1022.614,236.837,375.332,169.491,48.919,159.335
C01387=1022.607,236.589,375.360,169.487,48.923,159.336
C01388=1022.601,236.341,375.387,169.482,48.928,159.336
C01389=1022.595,236.092,375.414,169.479,48.932,159.336
C01390=1022.588,235.844,375.442,169.475,48.936,159.337
C01391=1022.582,235.595,375.469,169.471,48.940,159.337
C01392=1022.575,235.347,375.496,169.467,48.944,159.337
C01393=1022.569,235.099,375.524,169.464,48.948,159.338
C01394=1022.564,234.887,375.547,169.461,48.952,159.338
C01395=1022.558,234.675,375.571,169.458,48.955,159.338
C01396=1022.553,234.462,375.595,169.454,48.958,159.338
C01397=1022.547,234.251,375.617,169.451,48.962,159.339
C01398=1022.542,234.039,375.641,169.448,48.965,159.339
C01399=1022.536,233.827,375.664,169.444,48.969,159.339
C01400=1022.532,233.615,375.687,169.442,48.973,159.340
C01401=1022.526,233.403,375.711,169.439,48.976,159.340
C01402=1022.520,233.155,375.738,169.435,48.980,159.340
C01403=1022.514,232.906,375.766,169.431,48.984,159.341
C01404=1022.507,232.658,375.793,169.428,48.989,159.341
C01405=1022.501,232.409,375.820,169.424,48.993,159.341
C01406=1022.494,232.161,375.848,169.420,48.997,159.342
C01407=1022.489,231.913,375.874,169.417,49.001,159.342
C01408=1022.482,231.664,375.902,169.413,49.005,159.342
C01409=1022.476,231.416,375.929,169.408,49.010,159.343
C01410=1022.470,231.167,375.956,169.405,49.014,159.343
C01411=1022.463,230.918,375.983,169.401,49.018,159.343
C01412=1022.457,230.671,376.011,169.397,49.022,159.344
C01413=1022.451,230.421,376.038,169.394,49.027,159.344
C01414=1022.445,230.174,376.065,169.390,49.031,159.345
C01415=1022.438,229.925,376.092,169.386,49.035,159.345
C01416=1022.432,229.676,376.119,169.383,49.040,159.345
C01417=1022.426,229.428,376.147,169.380,49.044,159.346
C01418=1022.420,229.180,376.173,169.376,49.048,159.346
C01419=1022.413,228.931,376.201,169.372,49.052,159.346
C01420=1022.408,228.683,376.228,169.369,49.057,159.347
C01421=1022.400,228.434,376.254,169.365,49.061,159.347
C01422=1022.394,228.186,376.281,169.362,49.066,159.348
C01423=1022.388,227.937,376.308,169.358,49.070,159.348
C01424=1022.382,227.689,376.335,169.354,49.074,159.348
C01425=1022.376,227.440,376.363,169.351,49.078,159.349
C01426=1022.370,227.192,376.389,169.347,49.082,159.349
C01427=1022.363,226.943,376.416,169.343,49.087,159.350
C01428=1022.357,226.695,376.443,169.339,49.092,159.350
C01429=1022.350,226.446,376.470,169.335,49.096,159.350
C01430=1022.344,226.198,376.497,169.332,49.101,159.351
C01431=1022.337,225.949,376.523,169.328,49.105,159.351
C01432=1022.332,225.701,376.550,169.325,49.109,159.352
C01433=1022.325,225.452,376.577,169.321,49.114,159.352
C01434=1022.319,225.204,376.603,169.318,49.118,159.352
C01435=1022.312,224.955,376.630,169.314,49.122,159.353
C01436=1022.306,224.706,376.657,169.310,49.128,159.353
C01437=1022.299,224.458,376.684,169.306,49.132,159.354
C01438=1022.293,224.210,376.710,169.303,49.137,159.354
C01439=1022.288,223.962,376.737,169.299,49.141,159.354
C01440=1022.280,223.713,376.764,169.296,49.145,159.355
C01441=1022.275,223.465,376.790,169.292,49.150,159.355
C01442=1022.268,223.216,376.817,169.289,49.154,159.356
C01443=1022.262,222.967,376.843,169.285,49.159,159.356
C01444=1022.255,222.718,376.870,169.282,49.163,159.357
C01445=1022.249,222.470,376.896,169.277,49.168,159.357
C01446=1022.243,222.222,376.923,169.274,49.173,159.357
C01447=1022.237,221.973,376.950,169.270,49.177,159.358
C01448=1022.230,221.725,376.976,169.267,49.182,159.358
C01449=1022.224,221.476,377.003,169.263,49.186,159.359
C01450=1022.218,221.227,377.030,169.260,49.191,159.359
C01451=1022.212,220.979,377.056,169.256,49.195,159.359
C01452=1022.205,220.730,377.083,169.253,49.200,159.360
C01453=1022.199,220.482,377.109,169.249,49.204,159.360
C01454=1022.194,220.266,377.131,169.246,49.208,159.361
C01455=1022.188,220.050,377.155,169.243,49.212,159.361
C01456=1022.183,219.834,377.178,169.239,49.216,159.362
C01457=1022.178,219.618,377.201,169.237,49.220,159.362
C01458=1022.172,219.402,377.224,169.234,49.224,159.362
C01459=1022.167,219.187,377.247,169.230,49.228,159.363
C01460=1022.162,218.971,377.270,169.228,49.232,159.363
C01461=1022.155,218.755,377.293,169.224,49.236,159.363
C01462=1022.150,218.506,377.320,169.221,49.241,159.364
C01463=1022.143,218.258,377.346,169.217,49.246,159.364
C01464=1022.137,218.009,377.372,169.214,49.250,159.365
C01465=1022.131,217.761,377.398,169.211,49.255,159.365
C01466=1022.124,217.513,377.424,169.206,49.260,159.366
C01467=1022.118,217.264,377.451,169.203,49.265,159.366
C01468=1022.111,217.015,377.476,169.199,49.270,159.367
C01469=1022.105,216.767,377.502,169.196,49.274,159.367
C01470=1022.099,216.518,377.529,169.193,49.279,159.368
C01471=1022.092,216.269,377.555,169.189,49.284,159.368
C01472=1022.086,216.021,377.581,169.185,49.289,159.369
C01473=1022.080,215.773,377.608,169.182,49.294,159.369
C01474=1022.074,215.524,377.633,169.178,49.299,159.370
C01475=1022.067,215.275,377.659,169.175,49.303,159.370
C01476=1022.061,215.027,377.686,169.171,49.308,159.371
C01477=1022.055,214.778,377.711,169.168,49.313,159.371
C01478=1022.048,214.529,377.738,169.164,49.318,159.372
C01479=1022.042,214.280,377.764,169.161,49.323,159.372
C01480=1022.036,214.032,377.790,169.157,49.327,159.373
C01481=1022.029,213.784,377.816,169.154,49.332,159.373
C01482=1022.024,213.535,377.842,169.150,49.337,159.374
C01483=1022.017,213.287,377.868,169.147,49.342,159.374
C01484=1022.010,213.038,377.893,169.143,49.347,159.375
C01485=1022.005,212.790,377.920,169.139,49.352,159.375
C01486=1021.998,212.541,377.945,169.136,49.357,159.376
C01487=1021.991,212.292,377.972,169.133,49.361,159.376
C01488=1021.986,212.043,377.998,169.129,49.366,159.377
C01489=1021.979,211.795,378.024,169.126,49.371,159.377
C01490=1021.973,211.546,378.049,169.123,49.375,159.378
C01491=1021.967,211.298,378.076,169.118,49.381,159.378
C01492=1021.961,211.049,378.101,169.115,49.386,159.379
C01493=1021.954,210.801,378.128,169.112,49.390,159.379
C01494=1021.949,210.552,378.153,169.109,49.395,159.380
C01495=1021.942,210.304,378.180,169.105,49.400,159.380
C01496=1021.936,210.055,378.205,169.102,49.405,159.381
C01497=1021.929,209.807,378.231,169.098,49.410,159.381
C01498=1021.924,209.558,378.257,169.094,49.415,159.382
C01499=1021.918,209.309,378.282,169.091,49.420,159.382
C01500=1021.910,209.060,378.309,169.088,49.425,159.383
C01501=1021.904,208.812,378.334,169.085,49.430,159.383
C01502=1021.898,208.563,378.359,169.080,49.435,159.384
C01503=1021.892,208.315,378.385,169.077,49.440,159.384
C01504=1021.885,208.066,378.411,169.074,49.445,159.385
C01505=1021.880,207.817,378.437,169.071,49.451,159.386
C01506=1021.873,207.569,378.463,169.067,49.456,159.386
C01507=1021.867,207.321,378.488,169.063,49.461,159.387
C01508=1021.860,207.071,378.514,169.060,49.466,159.387
C01509=1021.854,206.823,378.539,169.057,49.471,159.388
C01510=1021.848,206.575,378.565,169.054,49.475,159.388
C01511=1021.841,206.326,378.590,169.050,49.481,159.389
C01512=1021.835,206.077,378.616,169.046,49.486,159.389
C01513=1021.829,205.829,378.641,169.043,49.491,159.390
C01514=1021.824,205.614,378.663,169.040,49.495,159.390
C01515=1021.818,205.401,378.685,169.037,49.500,159.391
C01516=1021.813,205.187,378.708,169.034,49.504,159.391
C01517=1021.807,204.974,378.729,169.031,49.509,159.392
C01518=1021.802,204.759,378.751,169.028,49.514,159.392
C01519=1021.796,204.545,378.773,169.026,49.518,159.393
C01520=1021.791,204.331,378.795,169.022,49.523,159.393
C01521=1021.763,203.081,378.916,168.586,49.431,159.305
C01522=1021.757,202.833,378.940,168.581,49.437,159.306
C01523=1021.751,202.584,378.964,168.577,49.443,159.306
C01524=1021.746,202.335,378.987,168.573,49.449,159.307
C01525=1021.741,202.087,379.012,168.569,49.456,159.308
C01526=1021.735,201.838,379.035,168.565,49.462,159.308
C01527=1021.730,201.589,379.059,168.560,49.468,159.309
C01528=1021.725,201.340,379.083,168.556,49.474,159.310
C01529=1021.719,201.092,379.106,168.552,49.480,159.310
C01530=1021.714,200.843,379.130,168.547,49.486,159.311
C01531=1021.709,200.594,379.154,168.543,49.492,159.311
C01532=1021.704,200.345,379.178,168.539,49.498,159.312
C01533=1021.698,200.096,379.201,168.534,49.504,159.312
C01534=1021.692,199.847,379.226,168.530,49.511,159.313
C01535=1021.687,199.598,379.249,168.526,49.517,159.314
C01536=1021.681,199.349,379.273,168.521,49.523,159.314
C01537=1021.676,199.100,379.296,168.517,49.529,159.315
C01538=1021.670,198.851,379.319,168.513,49.536,159.316
C01539=1021.664,198.603,379.343,168.509,49.542,159.316
C01540=1021.659,198.354,379.367,168.505,49.548,159.317
C01541=1021.653,198.105,379.390,168.500,49.555,159.317
C01542=1021.647,197.857,379.413,168.496,49.560,159.318
C01543=1021.642,197.608,379.437,168.491,49.567,159.319
C01544=1021.637,197.359,379.460,168.488,49.573,159.319
C01545=1021.632,197.109,379.483,168.484,49.579,159.320
C01546=1021.626,196.861,379.507,168.479,49.586,159.320
C01547=1021.620,196.612,379.530,168.475,49.591,159.321
C01548=1021.615,196.363,379.553,168.471,49.598,159.322
C01549=1021.609,196.114,379.576,168.466,49.604,159.322
C01550=1021.603,195.865,379.599,168.462,49.610,159.323
C01551=1021.598,195.617,379.624,168.459,49.617,159.324
C01552=1021.592,195.368,379.646,168.454,49.623,159.324
C01553=1021.587,195.119,379.669,168.450,49.629,159.325
C01554=1021.582,194.870,379.693,168.446,49.636,159.326
C01555=1021.576,194.621,379.716,168.441,49.642,159.326
C01556=1021.571,194.373,379.738,168.438,49.648,159.327
C01557=1021.565,194.124,379.763,168.434,49.655,159.328
C01558=1021.560,193.875,379.786,168.429,49.661,159.328
C01559=1021.555,193.626,379.809,168.425,49.667,159.329
C01560=1021.549,193.377,379.832,168.421,49.673,159.329
C01561=1021.543,193.128,379.855,168.417,49.680,159.330
C01562=1021.538,192.879,379.879,168.413,49.686,159.331
C01563=1021.533,192.631,379.901,168.409,49.692,159.331
C01564=1021.527,192.382,379.924,168.405,49.698,159.332
C01565=1021.522,192.133,379.948,168.401,49.705,159.333
C01566=1021.517,191.884,379.971,168.397,49.711,159.333
C01567=1021.511,191.635,379.994,168.393,49.717,159.334
C01568=1021.506,191.386,380.017,168.388,49.724,159.334
C01569=1021.500,191.137,380.040,168.384,49.730,159.335
C01570=1021.495,190.888,380.063,168.380,49.736,159.336
C01571=1021.490,190.639,380.086,168.377,49.743,159.336
C01572=1021.484,190.390,380.109,168.372,49.749,159.337
C01573=1021.479,190.141,380.132,168.368,49.755,159.338
C01574=1021.474,189.892,380.156,168.364,49.762,159.338
C01575=1021.469,189.644,380.178,168.360,49.768,159.339
C01576=1021.463,189.395,380.201,168.357,49.774,159.340
C01577=1021.458,189.146,380.225,168.352,49.780,159.340
C01578=1021.452,188.897,380.248,168.348,49.786,159.341
C01579=1021.447,188.649,380.270,168.344,49.793,159.342
C01580=1021.442,188.400,380.294,168.340,49.799,159.342
C01581=1021.436,188.151,380.317,168.336,49.805,159.343
C01582=1021.431,187.869,380.342,168.332,49.813,159.344
C01583=1021.425,187.587,380.368,168.328,49.820,159.344
C01584=1021.418,187.306,380.395,168.323,49.827,159.345
C01585=1021.413,187.024,380.420,168.319,49.834,159.346
C01586=1021.407,186.775,380.443,168.314,49.841,159.346
C01587=1021.402,186.527,380.466,168.310,49.847,159.347
C01588=1021.397,186.278,380.489,168.306,49.853,159.348
C01589=1021.391,186.029,380.512,168.303,49.859,159.348
C01590=1021.386,185.780,380.535,168.299,49.865,159.349
C01591=1021.381,185.531,380.557,168.295,49.872,159.350
C01592=1021.376,185.282,380.580,168.290,49.878,159.350
C01593=1021.370,185.033,380.603,168.286,49.884,159.351
C01594=1021.366,184.784,380.627,168.283,49.891,159.352
C01595=1021.360,184.535,380.649,168.279,49.897,159.352
C01596=1021.355,184.287,380.671,168.275,49.903,159.353
C01597=1021.350,184.037,380.695,168.271,49.909,159.354
C01598=1021.344,183.789,380.718,168.267,49.915,159.354
C01599=1021.339,183.540,380.740,168.264,49.922,159.355
C01600=1021.335,183.290,380.763,168.260,49.928,159.356
C01601=1021.329,183.042,380.786,168.255,49.934,159.356
C01602=1021.324,182.793,380.808,168.252,49.941,159.357
C01603=1021.319,182.544,380.832,168.248,49.947,159.357
C01604=1021.313,182.295,380.855,168.244,49.954,159.358
C01605=1021.308,182.046,380.876,168.240,49.960,159.359
C01606=1021.303,181.796,380.899,168.237,49.966,159.360
C01607=1021.297,181.548,380.921,168.233,49.973,159.360
C01608=1021.292,181.299,380.943,168.228,49.979,159.361
C01609=1021.286,181.050,380.966,168.225,49.986,159.362
C01610=1021.280,180.801,380.987,168.221,49.993,159.362
C01611=1021.275,180.552,381.009,168.217,49.999,159.363
C01612=1021.269,180.303,381.032,168.213,50.006,159.364
C01613=1021.263,180.054,381.054,168.209,50.013,159.365
C01614=1021.258,179.805,381.076,168.206,50.019,159.365
C01615=1021.253,179.556,381.098,168.202,50.025,159.366
C01616=1021.247,179.308,381.120,168.198,50.032,159.367
C01617=1021.242,179.058,381.142,168.194,50.039,159.367
C01618=1021.236,178.809,381.164,168.190,50.045,159.368
C01619=1021.231,178.560,381.187,168.186,50.052,159.369
C01620=1021.225,178.311,381.209,168.183,50.058,159.370
C01621=1021.220,178.062,381.230,168.179,50.065,159.370
C01622=1021.215,177.813,381.253,168.174,50.071,159.371
C01623=1021.209,177.565,381.275,168.171,50.078,159.372
C01624=1021.203,177.316,381.297,168.167,50.085,159.372
C01625=1021.198,177.066,381.319,168.163,50.091,159.373
C01626=1021.192,176.818,381.340,168.160,50.098,159.374
C01627=1021.187,176.568,381.363,168.156,50.104,159.374
C01628=1021.182,176.320,381.385,168.152,50.111,159.375
C01629=1021.176,176.071,381.407,168.148,50.117,159.376
C01630=1021.171,175.822,381.429,168.144,50.124,159.377
C01631=1021.165,175.572,381.451,168.141,50.131,159.377
C01632=1021.160,175.324,381.472,168.137,50.137,159.378
C01633=1021.154,175.074,381.494,168.134,50.144,159.379
C01634=1021.150,174.825,381.516,168.130,50.150,159.379
C01635=1021.143,174.577,381.539,168.127,50.157,159.380
C01636=1021.138,174.328,381.561,168.122,50.163,159.381
C01637=1021.133,174.079,381.583,168.118,50.170,159.382
C01638=1021.127,173.830,381.604,168.115,50.177,159.382
C01639=1021.122,173.580,381.626,168.111,50.183,159.383
C01640=1021.117,173.332,381.648,168.107,50.189,159.384
C01641=1021.111,173.083,381.669,168.104,50.196,159.384
C01642=1021.106,172.834,381.692,168.100,50.203,159.385
C01643=1021.101,172.585,381.714,168.096,50.209,159.386
C01644=1021.095,172.336,381.735,168.093,50.216,159.387
C01645=1021.090,172.087,381.757,168.089,50.222,159.387
C01646=1021.083,171.805,381.782,168.085,50.229,159.388
C01647=1021.078,171.523,381.806,168.081,50.237,159.389
C01648=1021.072,171.240,381.832,168.077,50.245,159.390
C01649=1021.066,170.958,381.856,168.072,50.252,159.391
C01650=1021.061,170.710,381.878,168.069,50.259,159.391
C01651=1021.055,170.460,381.899,168.065,50.265,159.392
C01652=1021.050,170.212,381.921,168.061,50.272,159.393
C01653=1021.045,169.962,381.943,168.058,50.278,159.393
C01654=1021.039,169.713,381.965,168.054,50.285,159.394
C01655=1021.034,169.465,381.986,168.051,50.292,159.395
C01656=1021.029,169.215,382.009,168.047,50.298,159.396
C01657=1021.023,168.967,382.030,168.043,50.305,159.396
C01658=1021.018,168.718,382.052,168.040,50.311,159.397
C01659=1021.013,168.468,382.074,168.036,50.317,159.398
C01660=1021.007,168.220,382.095,168.033,50.324,159.399
C01661=1021.003,167.971,382.117,168.029,50.331,159.399
C01662=1020.997,167.721,382.139,168.025,50.337,159.400
C01663=1020.992,167.473,382.161,168.022,50.344,159.401
C01664=1020.987,167.224,382.182,168.018,50.350,159.401
C01665=1020.981,166.974,382.203,168.015,50.357,159.402
C01666=1020.976,166.726,382.225,168.011,50.363,159.403
C01667=1020.971,166.477,382.247,168.007,50.370,159.404
C01668=1020.966,166.228,382.268,168.004,50.377,159.404
C01669=1020.960,165.979,382.291,168.000,50.383,159.405
C01670=1020.956,165.729,382.312,167.997,50.390,159.406
C01671=1020.950,165.481,382.333,167.993,50.396,159.406
C01672=1020.945,165.231,382.355,167.990,50.403,159.407
C01673=1020.940,164.982,382.377,167.986,50.409,159.408
C01674=1020.934,164.734,382.398,167.982,50.416,159.409
C01675=1020.930,164.484,382.420,167.980,50.422,159.410
C01676=1020.924,164.235,382.441,167.976,50.428,159.410
C01677=1020.919,163.986,382.463,167.973,50.435,159.411
C01678=1020.914,163.738,382.485,167.969,50.442,159.412
C01679=1020.909,163.489,382.506,167.965,50.448,159.412
C01680=1020.904,163.240,382.527,167.962,50.455,159.413
C01681=1020.899,162.990,382.550,167.958,50.462,159.414
C01682=1020.893,162.742,382.571,167.955,50.468,159.414
C01683=1020.888,162.492,382.592,167.951,50.474,159.415
C01684=1020.883,162.244,382.613,167.948,50.481,159.416
C01685=1020.878,161.995,382.635,167.944,50.487,159.416
C01686=1020.873,161.745,382.657,167.941,50.494,159.417
C01687=1020.867,161.496,382.678,167.938,50.500,159.418
C01688=1020.863,161.247,382.700,167.934,50.507,159.419
C01689=1020.858,160.998,382.721,167.931,50.513,159.419
C01690=1020.853,160.750,382.742,167.927,50.520,159.420
C01691=1020.848,160.501,382.764,167.924,50.527,159.421
C01692=1020.842,160.251,382.785,167.920,50.533,159.422
C01693=1020.837,160.002,382.807,167.917,50.539,159.423
C01694=1020.832,159.753,382.829,167.914,50.546,159.423
C01695=1020.827,159.504,382.849,167.910,50.552,159.424
C01696=1020.822,159.255,382.871,167.907,50.559,159.425
C01697=1020.818,159.006,382.892,167.903,50.566,159.425
C01698=1020.812,158.757,382.914,167.899,50.572,159.426
C01699=1020.806,158.508,382.934,167.896,50.579,159.427
C01700=1020.801,158.259,382.956,167.892,50.586,159.428
C01701=1020.795,158.010,382.976,167.889,50.592,159.428
C01702=1020.791,157.760,382.997,167.886,50.599,159.429
C01703=1020.785,157.512,383.019,167.883,50.606,159.430
C01704=1020.780,157.263,383.039,167.880,50.612,159.431
C01705=1020.774,157.013,383.060,167.876,50.619,159.432
C01706=1020.769,156.765,383.081,167.873,50.626,159.432
C01707=1020.763,156.515,383.102,167.869,50.632,159.433
C01708=1020.759,156.266,383.123,167.866,50.639,159.434
C01709=1020.753,156.017,383.144,167.862,50.646,159.434
C01710=1020.748,155.735,383.168,167.858,50.653,159.435
C01711=1020.741,155.452,383.191,167.855,50.661,159.436
C01712=1020.735,155.170,383.215,167.851,50.669,159.437
C01713=1020.729,154.888,383.239,167.847,50.676,159.438
C01714=1020.724,154.639,383.259,167.843,50.683,159.439
C01715=1020.718,154.390,383.281,167.840,50.690,159.439
C01716=1020.713,154.141,383.301,167.836,50.696,159.440
C01717=1020.709,153.892,383.322,167.834,50.703,159.441
C01718=1020.703,153.642,383.343,167.830,50.710,159.442
C01719=1020.697,153.393,383.364,167.827,50.716,159.443
C01720=1020.692,153.144,383.385,167.824,50.723,159.443
C01721=1020.687,152.895,383.406,167.820,50.730,159.444
C01722=1020.681,152.646,383.426,167.817,50.737,159.445
C01723=1020.676,152.397,383.447,167.813,50.743,159.446
C01724=1020.671,152.148,383.467,167.809,50.750,159.446
C01725=1020.666,151.899,383.488,167.806,50.757,159.447
C01726=1020.660,151.650,383.509,167.804,50.763,159.448
C01727=1020.655,151.401,383.530,167.800,50.770,159.449
C01728=1020.650,151.152,383.550,167.797,50.777,159.449
C01729=1020.644,150.903,383.571,167.793,50.784,159.450
C01730=1020.639,150.654,383.591,167.790,50.790,159.451
C01731=1020.634,150.404,383.612,167.787,50.797,159.452
C01732=1020.629,150.155,383.632,167.783,50.804,159.453
C01733=1020.623,149.906,383.653,167.780,50.811,159.453
C01734=1020.618,149.657,383.673,167.777,50.817,159.454
C01735=1020.613,149.408,383.694,167.774,50.824,159.455
C01736=1020.608,149.159,383.715,167.771,50.831,159.456
C01737=1020.602,148.910,383.735,167.767,50.838,159.457
C01738=1020.597,148.661,383.756,167.764,50.845,159.457
C01739=1020.592,148.411,383.776,167.760,50.851,159.458
C01740=1020.587,148.162,383.797,167.757,50.858,159.459
C01741=1020.581,147.913,383.817,167.754,50.864,159.460
C01742=1020.576,147.664,383.838,167.751,50.871,159.460
C01743=1020.571,147.415,383.858,167.747,50.878,159.461
C01744=1020.566,147.166,383.879,167.744,50.885,159.462
C01745=1020.560,146.917,383.900,167.741,50.891,159.463
C01746=1020.555,146.668,383.920,167.737,50.898,159.463
C01747=1020.550,146.418,383.941,167.735,50.905,159.464
C01748=1020.544,146.170,383.961,167.731,50.912,159.465
C01749=1020.539,145.921,383.981,167.728,50.918,159.466
C01750=1020.533,145.671,384.002,167.725,50.925,159.467
C01751=1020.528,145.422,384.022,167.721,50.932,159.467
C01752=1020.523,145.173,384.042,167.718,50.939,159.468
C01753=1020.517,144.924,384.062,167.714,50.946,159.469
C01754=1020.512,144.675,384.083,167.712,50.952,159.470
C01755=1020.507,144.425,384.103,167.709,50.959,159.471
C01756=1020.502,144.176,384.123,167.705,50.966,159.471
C01757=1020.496,143.928,384.143,167.702,50.973,159.472
C01758=1020.491,143.678,384.163,167.698,50.980,159.473
C01759=1020.486,143.429,384.184,167.695,50.987,159.474
C01760=1020.480,143.180,384.203,167.692,50.993,159.475
C01761=1020.475,142.931,384.224,167.689,51.000,159.475
C01762=1020.469,142.682,384.244,167.686,51.007,159.476
C01763=1020.464,142.433,384.265,167.683,51.014,159.477
C01764=1020.459,142.183,384.284,167.679,51.021,159.478
C01765=1020.453,141.934,384.304,167.676,51.027,159.479
C01766=1020.449,141.686,384.325,167.673,51.034,159.479
C01767=1020.443,141.436,384.344,167.670,51.041,159.480
C01768=1020.438,141.187,384.364,167.667,51.048,159.481
C01769=1020.432,140.938,384.385,167.663,51.055,159.482
C01770=1020.427,140.688,384.405,167.660,51.061,159.482
C01771=1020.421,140.439,384.425,167.658,51.068,159.483
C01772=1020.416,140.190,384.445,167.654,51.075,159.484
C01773=1020.412,139.941,384.465,167.651,51.082,159.485
C01774=1020.406,139.659,384.487,167.647,51.090,159.486
C01775=1020.399,139.377,384.510,167.644,51.097,159.487
C01776=1020.394,139.094,384.533,167.640,51.105,159.488
C01777=1020.388,138.812,384.556,167.637,51.113,159.489
C01778=1020.383,138.562,384.576,167.634,51.119,159.489
C01779=1020.377,138.313,384.596,167.630,51.126,159.490
C01780=1020.372,138.063,384.616,167.627,51.133,159.491
C01781=1020.366,137.814,384.636,167.624,51.140,159.492
C01782=1020.361,137.565,384.656,167.621,51.147,159.493
C01783=1020.356,137.316,384.676,167.618,51.154,159.493
C01784=1020.350,137.067,384.695,167.614,51.160,159.494
C01785=1020.345,136.818,384.715,167.611,51.167,159.495
C01786=1020.339,136.568,384.735,167.609,51.174,159.496
C01787=1020.334,136.319,384.755,167.605,51.181,159.497
C01788=1020.329,136.070,384.774,167.602,51.188,159.497
C01789=1020.324,135.821,384.795,167.599,51.195,159.498
C01790=1020.318,135.572,384.814,167.596,51.201,159.499
C01791=1020.313,135.323,384.835,167.593,51.208,159.500
C01792=1020.308,135.074,384.853,167.590,51.215,159.501
C01793=1020.303,134.824,384.873,167.586,51.222,159.501
C01794=1020.297,134.575,384.893,167.583,51.229,159.502
C01795=1020.292,134.326,384.913,167.581,51.236,159.503
C01796=1020.287,134.078,384.933,167.578,51.243,159.504
C01797=1020.282,133.828,384.952,167.574,51.250,159.505
C01798=1020.276,133.578,384.972,167.571,51.257,159.505
C01799=1020.270,133.330,384.992,167.569,51.263,159.506
C01800=1020.266,133.081,385.011,167.565,51.270,159.507
C01801=1020.260,132.831,385.030,167.562,51.277,159.508
C01802=1020.255,132.582,385.051,167.559,51.284,159.509
C01803=1020.249,132.333,385.070,167.556,51.290,159.510
C01804=1020.245,132.084,385.090,167.553,51.297,159.510
C01805=1020.239,131.835,385.110,167.550,51.304,159.511
C01806=1020.234,131.585,385.129,167.546,51.311,159.512
C01807=1020.229,131.336,385.148,167.544,51.318,159.513
C01808=1020.223,131.087,385.168,167.541,51.325,159.514
C01809=1020.218,130.838,385.188,167.537,51.331,159.514
